LIN {X 125.150,Y 42.862,Z -41.660,A 90.000,B 90.000,C 0.000} C_DIS
LIN {X 125.083,Y 42.862,Z -40.727,A 90.000,B 90.000,C 0.000} C_DIS
LIN {X 124.959,Y 42.862,Z -39.799,A 90.000,B 90.000,C 0.000} C_DIS
LIN {X 124.777,Y 42.862,Z -38.880,A 90.000,B 90.000,C 0.000} C_DIS
LIN {X 124.742,Y 42.862,Z -38.744,A 90.000,B 90.000,C 0.000} C_DIS
LIN {X 144.015,Y 42.862,Z -38.744,A 90.000,B 90.000,C 0.000} C_DIS
LIN {X 144.015,Y 42.862,Z -31.195,A 90.000,B 90.000,C 0.000} C_DIS
LIN {X 120.047,Y 42.862,Z -31.195,A 90.000,B 90.000,C 0.000} C_DIS
LIN {X 119.392,Y 42.862,Z -30.675,A 90.000,B 90.000,C 0.000} C_DIS
LIN {X 118.703,Y 42.862,Z -30.202,A 90.000,B 90.000,C 0.000} C_DIS
LIN {X 117.982,Y 42.862,Z -29.778,A 90.000,B 90.000,C 0.000} C_DIS
LIN {X 117.233,Y 42.862,Z -29.405,A 90.000,B 90.000,C 0.000} C_DIS
LIN {X 116.461,Y 42.862,Z -29.085,A 90.000,B 90.000,C 0.000} C_DIS
LIN {X 115.668,Y 42.862,Z -28.820,A 90.000,B 90.000,C 0.000} C_DIS
LIN {X 114.858,Y 42.862,Z -28.611,A 90.000,B 90.000,C 0.000} C_DIS
LIN {X 114.036,Y 42.862,Z -28.458,A 90.000,B 90.000,C 0.000} C_DIS
LIN {X 113.205,Y 42.862,Z -28.364,A 90.000,B 90.000,C 0.000} C_DIS
LIN {X 113.054,Y 42.862,Z -28.333,A 90.000,B 90.000,C 0.000} C_DIS
LIN {X 112.017,Y 42.862,Z -28.254,A 90.000,B 90.000,C 0.000} C_DIS
LIN {X 110.978,Y 42.862,Z -28.245,A 90.000,B 90.000,C 0.000} C_DIS
LIN {X 109.940,Y 42.862,Z -28.305,A 90.000,B 90.000,C 0.000} C_DIS
LIN {X 108.908,Y 42.862,Z -28.435,A 90.000,B 90.000,C 0.000} C_DIS
LIN {X 107.888,Y 42.862,Z -28.633,A 90.000,B 90.000,C 0.000} C_DIS
LIN {X 106.883,Y 42.862,Z -28.899,A 90.000,B 90.000,C 0.000} C_DIS
LIN {X 105.898,Y 42.862,Z -29.232,A 90.000,B 90.000,C 0.000} C_DIS
LIN {X 104.937,Y 42.862,Z -29.630,A 90.000,B 90.000,C 0.000} C_DIS
LIN {X 104.006,Y 42.862,Z -30.091,A 90.000,B 90.000,C 0.000} C_DIS
LIN {X 103.107,Y 42.862,Z -30.614,A 90.000,B 90.000,C 0.000} C_DIS
LIN {X 102.245,Y 42.862,Z -31.195,A 90.000,B 90.000,C 0.000} C_DIS
LIN {X -144.015,Y 42.862,Z -31.195,A 90.000,B 90.000,C 0.000} C_DIS
LIN {X -144.015,Y 42.862,Z -38.744,A 90.000,B 90.000,C 0.000} C_DIS
LIN {X 94.730,Y 42.862,Z -38.744,A 90.000,B 90.000,C 0.000} C_DIS
LIN {X 86.696,Y 42.862,Z -46.293,A 90.000,B 90.000,C 0.000} C_DIS
LIN {X 56.285,Y 42.862,Z -46.293,A 90.000,B 90.000,C 0.000} C_DIS
LIN {X 57.224,Y 42.862,Z -46.739,A 90.000,B 90.000,C 0.000} C_DIS
LIN {X 58.135,Y 42.862,Z -47.241,A 90.000,B 90.000,C 0.000} C_DIS
LIN {X 59.013,Y 42.862,Z -47.797,A 90.000,B 90.000,C 0.000} C_DIS
LIN {X 59.857,Y 42.862,Z -48.404,A 90.000,B 90.000,C 0.000} C_DIS
LIN {X 60.662,Y 42.862,Z -49.062,A 90.000,B 90.000,C 0.000} C_DIS
LIN {X 61.427,Y 42.862,Z -49.766,A 90.000,B 90.000,C 0.000} C_DIS
LIN {X 62.148,Y 42.862,Z -50.516,A 90.000,B 90.000,C 0.000} C_DIS
LIN {X 62.822,Y 42.862,Z -51.307,A 90.000,B 90.000,C 0.000} C_DIS
LIN {X 63.559,Y 42.862,Z -52.125,A 90.000,B 90.000,C 0.000} C_DIS
LIN {X 64.266,Y 42.862,Z -52.970,A 90.000,B 90.000,C 0.000} C_DIS
LIN {X 64.941,Y 42.862,Z -53.841,A 90.000,B 90.000,C 0.000} C_DIS
LIN {X 78.905,Y 42.862,Z -53.841,A 90.000,B 90.000,C 0.000} C_DIS
LIN {X 77.974,Y 42.862,Z -55.025,A 90.000,B 90.000,C 0.000} C_DIS
LIN {X 77.084,Y 42.862,Z -56.241,A 90.000,B 90.000,C 0.000} C_DIS
LIN {X 76.237,Y 42.862,Z -57.487,A 90.000,B 90.000,C 0.000} C_DIS
LIN {X 75.433,Y 42.862,Z -58.761,A 90.000,B 90.000,C 0.000} C_DIS
LIN {X 74.674,Y 42.862,Z -60.063,A 90.000,B 90.000,C 0.000} C_DIS
LIN {X 73.961,Y 42.862,Z -61.390,A 90.000,B 90.000,C 0.000} C_DIS
LIN {X 69.034,Y 42.862,Z -61.390,A 90.000,B 90.000,C 0.000} C_DIS
LIN {X 68.549,Y 42.862,Z -60.157,A 90.000,B 90.000,C 0.000} C_DIS
LIN {X 68.010,Y 42.862,Z -58.947,A 90.000,B 90.000,C 0.000} C_DIS
LIN {X 67.418,Y 42.862,Z -57.762,A 90.000,B 90.000,C 0.000} C_DIS
LIN {X 66.774,Y 42.862,Z -56.605,A 90.000,B 90.000,C 0.000} C_DIS
LIN {X 66.080,Y 42.862,Z -55.477,A 90.000,B 90.000,C 0.000} C_DIS
LIN {X 65.335,Y 42.862,Z -54.381,A 90.000,B 90.000,C 0.000} C_DIS
LIN {X 64.543,Y 42.862,Z -53.320,A 90.000,B 90.000,C 0.000} C_DIS
LIN {X 63.705,Y 42.862,Z -52.294,A 90.000,B 90.000,C 0.000} C_DIS
LIN {X 62.822,Y 42.862,Z -51.307,A 90.000,B 90.000,C 0.000} C_DIS
LIN {X 62.102,Y 42.862,Z -50.466,A 90.000,B 90.000,C 0.000} C_DIS
LIN {X 61.330,Y 42.862,Z -49.672,A 90.000,B 90.000,C 0.000} C_DIS
LIN {X 60.509,Y 42.862,Z -48.930,A 90.000,B 90.000,C 0.000} C_DIS
LIN {X 59.641,Y 42.862,Z -48.241,A 90.000,B 90.000,C 0.000} C_DIS
LIN {X 58.732,Y 42.862,Z -47.610,A 90.000,B 90.000,C 0.000} C_DIS
LIN {X 57.783,Y 42.862,Z -47.039,A 90.000,B 90.000,C 0.000} C_DIS
LIN {X 56.800,Y 42.862,Z -46.529,A 90.000,B 90.000,C 0.000} C_DIS
LIN {X 55.787,Y 42.862,Z -46.083,A 90.000,B 90.000,C 0.000} C_DIS
LIN {X 54.746,Y 42.862,Z -45.704,A 90.000,B 90.000,C 0.000} C_DIS
LIN {X 53.684,Y 42.862,Z -45.392,A 90.000,B 90.000,C 0.000} C_DIS
LIN {X 52.797,Y 42.862,Z -45.129,A 90.000,B 90.000,C 0.000} C_DIS
LIN {X 51.895,Y 42.862,Z -44.923,A 90.000,B 90.000,C 0.000} C_DIS
LIN {X 50.982,Y 42.862,Z -44.775,A 90.000,B 90.000,C 0.000} C_DIS
LIN {X 50.062,Y 42.862,Z -44.685,A 90.000,B 90.000,C 0.000} C_DIS
LIN {X 49.137,Y 42.862,Z -44.654,A 90.000,B 90.000,C 0.000} C_DIS
LIN {X 48.213,Y 42.862,Z -44.681,A 90.000,B 90.000,C 0.000} C_DIS
LIN {X 47.292,Y 42.862,Z -44.767,A 90.000,B 90.000,C 0.000} C_DIS
LIN {X 46.319,Y 42.862,Z -44.277,A 90.000,B 90.000,C 0.000} C_DIS
LIN {X 45.314,Y 42.862,Z -43.856,A 90.000,B 90.000,C 0.000} C_DIS
LIN {X 44.282,Y 42.862,Z -43.505,A 90.000,B 90.000,C 0.000} C_DIS
LIN {X 43.229,Y 42.862,Z -43.227,A 90.000,B 90.000,C 0.000} C_DIS
LIN {X 42.159,Y 42.862,Z -43.022,A 90.000,B 90.000,C 0.000} C_DIS
LIN {X 41.077,Y 42.862,Z -42.891,A 90.000,B 90.000,C 0.000} C_DIS
LIN {X 39.989,Y 42.862,Z -42.836,A 90.000,B 90.000,C 0.000} C_DIS
LIN {X 38.899,Y 42.862,Z -42.856,A 90.000,B 90.000,C 0.000} C_DIS
LIN {X 37.814,Y 42.862,Z -42.951,A 90.000,B 90.000,C 0.000} C_DIS
LIN {X 36.738,Y 42.862,Z -43.121,A 90.000,B 90.000,C 0.000} C_DIS
LIN {X 35.676,Y 42.862,Z -43.365,A 90.000,B 90.000,C 0.000} C_DIS
LIN {X 34.633,Y 42.862,Z -43.681,A 90.000,B 90.000,C 0.000} C_DIS
LIN {X 33.615,Y 42.862,Z -44.069,A 90.000,B 90.000,C 0.000} C_DIS
LIN {X 32.626,Y 42.862,Z -44.527,A 90.000,B 90.000,C 0.000} C_DIS
LIN {X 31.671,Y 42.862,Z -45.052,A 90.000,B 90.000,C 0.000} C_DIS
LIN {X 30.755,Y 42.862,Z -45.641,A 90.000,B 90.000,C 0.000} C_DIS
LIN {X 29.882,Y 42.862,Z -46.293,A 90.000,B 90.000,C 0.000} C_DIS
LIN {X -144.015,Y 42.862,Z -46.293,A 90.000,B 90.000,C 0.000} C_DIS
LIN {X -144.015,Y 42.862,Z -53.841,A 90.000,B 90.000,C 0.000} C_DIS
LIN {X 24.711,Y 42.862,Z -53.841,A 90.000,B 90.000,C 0.000} C_DIS
LIN {X 24.711,Y 42.862,Z -53.843,A 90.000,B 90.000,C 0.000} C_DIS
LIN {X 24.175,Y 42.862,Z -54.360,A 90.000,B 90.000,C 0.000} C_DIS
LIN {X 23.668,Y 42.862,Z -54.907,A 90.000,B 90.000,C 0.000} C_DIS
LIN {X 23.192,Y 42.862,Z -55.480,A 90.000,B 90.000,C 0.000} C_DIS
LIN {X 22.748,Y 42.862,Z -56.078,A 90.000,B 90.000,C 0.000} C_DIS
LIN {X 22.337,Y 42.862,Z -56.700,A 90.000,B 90.000,C 0.000} C_DIS
LIN {X 21.899,Y 42.862,Z -57.594,A 90.000,B 90.000,C 0.000} C_DIS
LIN {X 21.518,Y 42.862,Z -58.513,A 90.000,B 90.000,C 0.000} C_DIS
LIN {X 21.196,Y 42.862,Z -59.455,A 90.000,B 90.000,C 0.000} C_DIS
LIN {X 20.934,Y 42.862,Z -60.415,A 90.000,B 90.000,C 0.000} C_DIS
LIN {X 20.734,Y 42.862,Z -61.390,A 90.000,B 90.000,C 0.000} C_DIS
LIN {X -144.015,Y 42.862,Z -61.390,A 90.000,B 90.000,C 0.000} C_DIS
LIN {X -144.015,Y 42.862,Z -68.939,A 90.000,B 90.000,C 0.000} C_DIS
LIN {X -16.258,Y 42.862,Z -68.939,A 90.000,B 90.000,C 0.000} C_DIS
LIN {X -17.508,Y 42.862,Z -69.258,A 90.000,B 90.000,C 0.000} C_DIS
LIN {X -18.739,Y 42.862,Z -69.643,A 90.000,B 90.000,C 0.000} C_DIS
LIN {X -19.948,Y 42.862,Z -70.093,A 90.000,B 90.000,C 0.000} C_DIS
LIN {X -21.131,Y 42.862,Z -70.607,A 90.000,B 90.000,C 0.000} C_DIS
LIN {X -22.284,Y 42.862,Z -71.183,A 90.000,B 90.000,C 0.000} C_DIS
LIN {X -23.406,Y 42.862,Z -71.821,A 90.000,B 90.000,C 0.000} C_DIS
LIN {X -24.492,Y 42.862,Z -72.517,A 90.000,B 90.000,C 0.000} C_DIS
LIN {X -25.539,Y 42.862,Z -73.271,A 90.000,B 90.000,C 0.000} C_DIS
LIN {X -26.544,Y 42.862,Z -74.079,A 90.000,B 90.000,C 0.000} C_DIS
LIN {X -27.504,Y 42.862,Z -74.940,A 90.000,B 90.000,C 0.000} C_DIS
LIN {X -28.266,Y 42.862,Z -75.705,A 90.000,B 90.000,C 0.000} C_DIS
LIN {X -29.009,Y 42.862,Z -76.488,A 90.000,B 90.000,C 0.000} C_DIS
LIN {X -144.015,Y 42.862,Z -76.488,A 90.000,B 90.000,C 0.000} C_DIS
LIN {X -144.015,Y 42.862,Z -84.037,A 90.000,B 90.000,C 0.000} C_DIS
LIN {X -34.671,Y 42.862,Z -84.037,A 90.000,B 90.000,C 0.000} C_DIS
LIN {X -35.506,Y 42.862,Z -85.491,A 90.000,B 90.000,C 0.000} C_DIS
LIN {X -36.286,Y 42.862,Z -86.975,A 90.000,B 90.000,C 0.000} C_DIS
LIN {X -37.012,Y 42.862,Z -88.487,A 90.000,B 90.000,C 0.000} C_DIS
LIN {X -37.681,Y 42.862,Z -90.025,A 90.000,B 90.000,C 0.000} C_DIS
LIN {X -38.293,Y 42.862,Z -91.586,A 90.000,B 90.000,C 0.000} C_DIS
LIN {X -144.015,Y 42.862,Z -91.586,A 90.000,B 90.000,C 0.000} C_DIS
LIN {X -144.015,Y 42.862,Z -99.134,A 90.000,B 90.000,C 0.000} C_DIS
LIN {X -40.372,Y 42.862,Z -99.134,A 90.000,B 90.000,C 0.000} C_DIS
LIN {X -40.520,Y 42.862,Z -99.983,A 90.000,B 90.000,C 0.000} C_DIS
LIN {X -40.653,Y 42.862,Z -100.835,A 90.000,B 90.000,C 0.000} C_DIS
LIN {X -40.931,Y 42.862,Z -101.987,A 90.000,B 90.000,C 0.000} C_DIS
LIN {X -41.159,Y 42.862,Z -103.150,A 90.000,B 90.000,C 0.000} C_DIS
LIN {X -41.337,Y 42.862,Z -104.322,A 90.000,B 90.000,C 0.000} C_DIS
LIN {X -41.464,Y 42.862,Z -105.500,A 90.000,B 90.000,C 0.000} C_DIS
LIN {X -41.540,Y 42.862,Z -106.683,A 90.000,B 90.000,C 0.000} C_DIS
LIN {X -144.015,Y 42.862,Z -106.683,A 90.000,B 90.000,C 0.000} C_DIS
LIN {X -144.015,Y 42.862,Z -114.232,A 90.000,B 90.000,C 0.000} C_DIS
LIN {X -41.253,Y 42.862,Z -114.232,A 90.000,B 90.000,C 0.000} C_DIS
LIN {X -41.121,Y 42.862,Z -114.920,A 90.000,B 90.000,C 0.000} C_DIS
LIN {X -40.964,Y 42.862,Z -115.603,A 90.000,B 90.000,C 0.000} C_DIS
LIN {X -40.701,Y 42.862,Z -116.533,A 90.000,B 90.000,C 0.000} C_DIS
LIN {X -40.478,Y 42.862,Z -117.474,A 90.000,B 90.000,C 0.000} C_DIS
LIN {X -40.295,Y 42.862,Z -118.423,A 90.000,B 90.000,C 0.000} C_DIS
LIN {X -40.153,Y 42.862,Z -119.379,A 90.000,B 90.000,C 0.000} C_DIS
LIN {X -40.093,Y 42.862,Z -119.584,A 90.000,B 90.000,C 0.000} C_DIS
LIN {X -40.057,Y 42.862,Z -119.773,A 90.000,B 90.000,C 0.000} C_DIS
LIN {X -39.705,Y 42.862,Z -120.775,A 90.000,B 90.000,C 0.000} C_DIS
LIN {X -39.361,Y 42.862,Z -121.781,A 90.000,B 90.000,C 0.000} C_DIS
LIN {X -144.015,Y 42.862,Z -121.781,A 90.000,B 90.000,C 0.000} C_DIS
LIN {X -144.015,Y 42.862,Z -129.329,A 90.000,B 90.000,C 0.000} C_DIS
LIN {X -36.708,Y 42.862,Z -129.329,A 90.000,B 90.000,C 0.000} C_DIS
LIN {X -36.411,Y 42.862,Z -129.970,A 90.000,B 90.000,C 0.000} C_DIS
LIN {X -36.089,Y 42.862,Z -130.598,A 90.000,B 90.000,C 0.000} C_DIS
LIN {X -35.628,Y 42.862,Z -131.888,A 90.000,B 90.000,C 0.000} C_DIS
LIN {X -35.126,Y 42.862,Z -133.162,A 90.000,B 90.000,C 0.000} C_DIS
LIN {X -34.584,Y 42.862,Z -134.419,A 90.000,B 90.000,C 0.000} C_DIS
LIN {X -34.001,Y 42.862,Z -135.658,A 90.000,B 90.000,C 0.000} C_DIS
LIN {X -33.379,Y 42.862,Z -136.878,A 90.000,B 90.000,C 0.000} C_DIS
LIN {X -144.015,Y 42.862,Z -136.878,A 90.000,B 90.000,C 0.000} C_DIS
LIN {X -144.015,Y 42.862,Z -144.427,A 90.000,B 90.000,C 0.000} C_DIS
LIN {X -28.091,Y 42.862,Z -144.427,A 90.000,B 90.000,C 0.000} C_DIS
LIN {X -26.928,Y 42.862,Z -145.648,A 90.000,B 90.000,C 0.000} C_DIS
LIN {X -25.719,Y 42.862,Z -146.824,A 90.000,B 90.000,C 0.000} C_DIS
LIN {X -24.467,Y 42.862,Z -147.953,A 90.000,B 90.000,C 0.000} C_DIS
LIN {X -23.173,Y 42.862,Z -149.035,A 90.000,B 90.000,C 0.000} C_DIS
LIN {X -21.839,Y 42.862,Z -150.066,A 90.000,B 90.000,C 0.000} C_DIS
LIN {X -20.468,Y 42.862,Z -151.047,A 90.000,B 90.000,C 0.000} C_DIS
LIN {X -19.060,Y 42.862,Z -151.976,A 90.000,B 90.000,C 0.000} C_DIS
LIN {X -144.015,Y 42.862,Z -151.976,A 90.000,B 90.000,C 0.000} C_DIS
LIN {X -144.015,Y 42.862,Z -159.525,A 90.000,B 90.000,C 0.000} C_DIS
LIN {X 24.265,Y 42.862,Z -159.525,A 90.000,B 90.000,C 0.000} C_DIS
LIN {X 23.466,Y 42.862,Z -160.862,A 90.000,B 90.000,C 0.000} C_DIS
LIN {X 22.621,Y 42.862,Z -162.169,A 90.000,B 90.000,C 0.000} C_DIS
LIN {X 21.729,Y 42.862,Z -163.445,A 90.000,B 90.000,C 0.000} C_DIS
LIN {X 20.793,Y 42.862,Z -164.689,A 90.000,B 90.000,C 0.000} C_DIS
LIN {X 19.813,Y 42.862,Z -165.899,A 90.000,B 90.000,C 0.000} C_DIS
LIN {X 18.790,Y 42.862,Z -167.073,A 90.000,B 90.000,C 0.000} C_DIS
LIN {X -144.015,Y 42.862,Z -167.073,A 90.000,B 90.000,C 0.000} C_DIS
LIN {X -144.015,Y 42.862,Z -174.622,A 90.000,B 90.000,C 0.000} C_DIS
LIN {X 10.993,Y 42.862,Z -174.622,A 90.000,B 90.000,C 0.000} C_DIS
LIN {X 9.938,Y 42.862,Z -175.710,A 90.000,B 90.000,C 0.000} C_DIS
LIN {X 8.046,Y 42.862,Z -177.766,A 90.000,B 90.000,C 0.000} C_DIS
LIN {X 6.126,Y 42.862,Z -179.795,A 90.000,B 90.000,C 0.000} C_DIS
LIN {X 5.088,Y 42.862,Z -180.989,A 90.000,B 90.000,C 0.000} C_DIS
LIN {X 4.035,Y 42.862,Z -182.171,A 90.000,B 90.000,C 0.000} C_DIS
LIN {X -144.015,Y 42.862,Z -182.171,A 90.000,B 90.000,C 0.000} C_DIS
LIN {X -144.015,Y 42.862,Z -189.720,A 90.000,B 90.000,C 0.000} C_DIS
LIN {X -3.333,Y 42.862,Z -189.720,A 90.000,B 90.000,C 0.000} C_DIS
LIN {X -4.736,Y 42.862,Z -191.028,A 90.000,B 90.000,C 0.000} C_DIS
LIN {X -6.158,Y 42.862,Z -192.316,A 90.000,B 90.000,C 0.000} C_DIS
LIN {X -8.323,Y 42.862,Z -194.009,A 90.000,B 90.000,C 0.000} C_DIS
LIN {X -10.520,Y 42.862,Z -195.660,A 90.000,B 90.000,C 0.000} C_DIS
LIN {X -12.749,Y 42.862,Z -197.269,A 90.000,B 90.000,C 0.000} C_DIS
LIN {X -144.015,Y 42.862,Z -197.269,A 90.000,B 90.000,C 0.000} C_DIS
LIN {X -144.015,Y 42.862,Z -204.817,A 90.000,B 90.000,C 0.000} C_DIS
LIN {X -24.715,Y 42.862,Z -204.817,A 90.000,B 90.000,C 0.000} C_DIS
LIN {X -28.376,Y 42.862,Z -206.710,A 90.000,B 90.000,C 0.000} C_DIS
LIN {X -32.061,Y 42.862,Z -208.555,A 90.000,B 90.000,C 0.000} C_DIS
LIN {X -35.770,Y 42.862,Z -210.351,A 90.000,B 90.000,C 0.000} C_DIS
LIN {X -39.503,Y 42.862,Z -212.098,A 90.000,B 90.000,C 0.000} C_DIS
LIN {X -40.093,Y 42.862,Z -212.366,A 90.000,B 90.000,C 0.000} C_DIS
LIN {X -144.015,Y 42.862,Z -212.366,A 90.000,B 90.000,C 0.000} C_DIS
LIN {X -144.015,Y 42.862,Z -219.915,A 90.000,B 90.000,C 0.000} C_DIS
LIN {X -55.981,Y 42.862,Z -219.915,A 90.000,B 90.000,C 0.000} C_DIS
LIN {X -60.909,Y 42.862,Z -222.383,A 90.000,B 90.000,C 0.000} C_DIS
LIN {X -65.811,Y 42.862,Z -224.899,A 90.000,B 90.000,C 0.000} C_DIS
LIN {X -70.689,Y 42.862,Z -227.464,A 90.000,B 90.000,C 0.000} C_DIS
LIN {X -144.015,Y 42.862,Z -227.464,A 90.000,B 90.000,C 0.000} C_DIS
LIN {X -144.015,Y 42.862,Z -235.012,A 90.000,B 90.000,C 0.000} C_DIS
LIN {X -84.330,Y 42.862,Z -235.012,A 90.000,B 90.000,C 0.000} C_DIS
LIN {X -86.708,Y 42.862,Z -236.453,A 90.000,B 90.000,C 0.000} C_DIS
LIN {X -89.064,Y 42.862,Z -237.928,A 90.000,B 90.000,C 0.000} C_DIS
LIN {X -91.399,Y 42.862,Z -239.438,A 90.000,B 90.000,C 0.000} C_DIS
LIN {X -93.711,Y 42.862,Z -240.983,A 90.000,B 90.000,C 0.000} C_DIS
LIN {X -96.000,Y 42.862,Z -242.561,A 90.000,B 90.000,C 0.000} C_DIS
LIN {X -144.015,Y 42.862,Z -242.561,A 90.000,B 90.000,C 0.000} C_DIS
LIN {X -144.015,Y 42.862,Z -23.646,A 90.000,B 90.000,C 0.000} C_DIS
LIN {X 144.015,Y 42.862,Z -23.646,A 90.000,B 90.000,C 0.000} C_DIS
LIN {X 144.015,Y 42.862,Z -16.098,A 90.000,B 90.000,C 0.000} C_DIS
LIN {X -144.015,Y 42.862,Z -16.098,A 90.000,B 90.000,C 0.000} C_DIS
LIN {X -144.015,Y 42.862,Z -8.549,A 90.000,B 90.000,C 0.000} C_DIS
LIN {X 144.015,Y 42.862,Z -8.549,A 90.000,B 90.000,C 0.000} C_DIS
LIN {X 144.015,Y 42.862,Z -1.000,A 90.000,B 90.000,C 0.000} C_DIS
LIN {X -144.015,Y 42.862,Z -1.000,A 90.000,B 90.000,C 0.000} C_DIS
LIN {X -3.685,Y 42.862,Z -68.939,A 90.000,B 90.000,C 0.000} C_DIS
LIN {X 10.592,Y 42.862,Z -68.939,A 90.000,B 90.000,C 0.000} C_DIS
LIN {X 10.606,Y 42.862,Z -73.107,A 90.000,B 90.000,C 0.000} C_DIS
LIN {X 7.736,Y 42.862,Z -72.365,A 90.000,B 90.000,C 0.000} C_DIS
LIN {X 4.853,Y 42.862,Z -71.676,A 90.000,B 90.000,C 0.000} C_DIS
LIN {X 1.958,Y 42.862,Z -71.039,A 90.000,B 90.000,C 0.000} C_DIS
LIN {X -0.948,Y 42.862,Z -70.455,A 90.000,B 90.000,C 0.000} C_DIS
LIN {X -3.864,Y 42.862,Z -69.924,A 90.000,B 90.000,C 0.000} C_DIS
LIN {X -4.992,Y 42.862,Z -69.694,A 90.000,B 90.000,C 0.000} C_DIS
LIN {X -6.128,Y 42.862,Z -69.514,A 90.000,B 90.000,C 0.000} C_DIS
LIN {X -7.272,Y 42.862,Z -69.383,A 90.000,B 90.000,C 0.000} C_DIS
LIN {X -8.420,Y 42.862,Z -69.302,A 90.000,B 90.000,C 0.000} C_DIS
LIN {X -9.570,Y 42.862,Z -69.272,A 90.000,B 90.000,C 0.000} C_DIS
LIN {X -10.721,Y 42.862,Z -69.292,A 90.000,B 90.000,C 0.000} C_DIS
LIN {X -11.870,Y 42.862,Z -69.361,A 90.000,B 90.000,C 0.000} C_DIS
LIN {X -13.141,Y 42.862,Z -69.448,A 90.000,B 90.000,C 0.000} C_DIS
LIN {X -14.406,Y 42.862,Z -69.605,A 90.000,B 90.000,C 0.000} C_DIS
LIN {X -15.659,Y 42.862,Z -69.832,A 90.000,B 90.000,C 0.000} C_DIS
LIN {X -16.899,Y 42.862,Z -70.127,A 90.000,B 90.000,C 0.000} C_DIS
LIN {X -18.120,Y 42.862,Z -70.490,A 90.000,B 90.000,C 0.000} C_DIS
LIN {X -19.320,Y 42.862,Z -70.919,A 90.000,B 90.000,C 0.000} C_DIS
LIN {X -20.494,Y 42.862,Z -71.414,A 90.000,B 90.000,C 0.000} C_DIS
LIN {X -21.639,Y 42.862,Z -71.973,A 90.000,B 90.000,C 0.000} C_DIS
LIN {X -22.752,Y 42.862,Z -72.594,A 90.000,B 90.000,C 0.000} C_DIS
LIN {X -23.828,Y 42.862,Z -73.276,A 90.000,B 90.000,C 0.000} C_DIS
LIN {X -24.866,Y 42.862,Z -74.015,A 90.000,B 90.000,C 0.000} C_DIS
LIN {X -25.861,Y 42.862,Z -74.811,A 90.000,B 90.000,C 0.000} C_DIS
LIN {X -26.811,Y 42.862,Z -75.660,A 90.000,B 90.000,C 0.000} C_DIS
LIN {X -28.077,Y 42.862,Z -76.954,A 90.000,B 90.000,C 0.000} C_DIS
LIN {X -29.289,Y 42.862,Z -78.298,A 90.000,B 90.000,C 0.000} C_DIS
LIN {X -30.445,Y 42.862,Z -79.690,A 90.000,B 90.000,C 0.000} C_DIS
LIN {X -31.543,Y 42.862,Z -81.128,A 90.000,B 90.000,C 0.000} C_DIS
LIN {X -32.583,Y 42.862,Z -82.610,A 90.000,B 90.000,C 0.000} C_DIS
LIN {X -33.561,Y 42.862,Z -84.132,A 90.000,B 90.000,C 0.000} C_DIS
LIN {X -34.476,Y 42.862,Z -85.694,A 90.000,B 90.000,C 0.000} C_DIS
LIN {X -35.327,Y 42.862,Z -87.291,A 90.000,B 90.000,C 0.000} C_DIS
LIN {X -36.112,Y 42.862,Z -88.922,A 90.000,B 90.000,C 0.000} C_DIS
LIN {X -36.830,Y 42.862,Z -90.583,A 90.000,B 90.000,C 0.000} C_DIS
LIN {X -37.480,Y 42.862,Z -92.272,A 90.000,B 90.000,C 0.000} C_DIS
LIN {X -38.060,Y 42.862,Z -93.986,A 90.000,B 90.000,C 0.000} C_DIS
LIN {X -38.570,Y 42.862,Z -95.723,A 90.000,B 90.000,C 0.000} C_DIS
LIN {X -39.009,Y 42.862,Z -97.478,A 90.000,B 90.000,C 0.000} C_DIS
LIN {X -39.377,Y 42.862,Z -99.250,A 90.000,B 90.000,C 0.000} C_DIS
LIN {X -39.671,Y 42.862,Z -101.036,A 90.000,B 90.000,C 0.000} C_DIS
LIN {X -39.961,Y 42.862,Z -102.237,A 90.000,B 90.000,C 0.000} C_DIS
LIN {X -40.195,Y 42.862,Z -103.450,A 90.000,B 90.000,C 0.000} C_DIS
LIN {X -40.372,Y 42.862,Z -104.673,A 90.000,B 90.000,C 0.000} C_DIS
LIN {X -40.492,Y 42.862,Z -105.902,A 90.000,B 90.000,C 0.000} C_DIS
LIN {X -40.555,Y 42.862,Z -107.136,A 90.000,B 90.000,C 0.000} C_DIS
LIN {X -40.560,Y 42.862,Z -108.372,A 90.000,B 90.000,C 0.000} C_DIS
LIN {X -40.508,Y 42.862,Z -109.606,A 90.000,B 90.000,C 0.000} C_DIS
LIN {X -40.546,Y 42.862,Z -110.568,A 90.000,B 90.000,C 0.000} C_DIS
LIN {X -40.534,Y 42.862,Z -111.530,A 90.000,B 90.000,C 0.000} C_DIS
LIN {X -40.474,Y 42.862,Z -112.491,A 90.000,B 90.000,C 0.000} C_DIS
LIN {X -40.364,Y 42.862,Z -113.447,A 90.000,B 90.000,C 0.000} C_DIS
LIN {X -40.206,Y 42.862,Z -114.397,A 90.000,B 90.000,C 0.000} C_DIS
LIN {X -40.000,Y 42.862,Z -115.337,A 90.000,B 90.000,C 0.000} C_DIS
LIN {X -39.734,Y 42.862,Z -116.283,A 90.000,B 90.000,C 0.000} C_DIS
LIN {X -39.506,Y 42.862,Z -117.238,A 90.000,B 90.000,C 0.000} C_DIS
LIN {X -39.319,Y 42.862,Z -118.203,A 90.000,B 90.000,C 0.000} C_DIS
LIN {X -39.171,Y 42.862,Z -119.174,A 90.000,B 90.000,C 0.000} C_DIS
LIN {X -39.119,Y 42.862,Z -119.351,A 90.000,B 90.000,C 0.000} C_DIS
LIN {X -39.089,Y 42.862,Z -119.511,A 90.000,B 90.000,C 0.000} C_DIS
LIN {X -38.572,Y 42.862,Z -120.993,A 90.000,B 90.000,C 0.000} C_DIS
LIN {X -38.075,Y 42.862,Z -122.483,A 90.000,B 90.000,C 0.000} C_DIS
LIN {X -37.597,Y 42.862,Z -123.978,A 90.000,B 90.000,C 0.000} C_DIS
LIN {X -37.537,Y 42.862,Z -124.124,A 90.000,B 90.000,C 0.000} C_DIS
LIN {X -37.324,Y 42.862,Z -124.797,A 90.000,B 90.000,C 0.000} C_DIS
LIN {X -37.062,Y 42.862,Z -125.453,A 90.000,B 90.000,C 0.000} C_DIS
LIN {X -36.753,Y 42.862,Z -126.088,A 90.000,B 90.000,C 0.000} C_DIS
LIN {X -36.523,Y 42.862,Z -126.941,A 90.000,B 90.000,C 0.000} C_DIS
LIN {X -36.248,Y 42.862,Z -127.780,A 90.000,B 90.000,C 0.000} C_DIS
LIN {X -35.931,Y 42.862,Z -128.604,A 90.000,B 90.000,C 0.000} C_DIS
LIN {X -35.571,Y 42.862,Z -129.411,A 90.000,B 90.000,C 0.000} C_DIS
LIN {X -35.169,Y 42.862,Z -130.197,A 90.000,B 90.000,C 0.000} C_DIS
LIN {X -34.647,Y 42.862,Z -131.656,A 90.000,B 90.000,C 0.000} C_DIS
LIN {X -34.070,Y 42.862,Z -133.095,A 90.000,B 90.000,C 0.000} C_DIS
LIN {X -33.441,Y 42.862,Z -134.511,A 90.000,B 90.000,C 0.000} C_DIS
LIN {X -32.759,Y 42.862,Z -135.903,A 90.000,B 90.000,C 0.000} C_DIS
LIN {X -32.026,Y 42.862,Z -137.269,A 90.000,B 90.000,C 0.000} C_DIS
LIN {X -31.243,Y 42.862,Z -138.606,A 90.000,B 90.000,C 0.000} C_DIS
LIN {X -30.411,Y 42.862,Z -139.914,A 90.000,B 90.000,C 0.000} C_DIS
LIN {X -29.530,Y 42.862,Z -141.189,A 90.000,B 90.000,C 0.000} C_DIS
LIN {X -28.431,Y 42.862,Z -142.533,A 90.000,B 90.000,C 0.000} C_DIS
LIN {X -27.280,Y 42.862,Z -143.832,A 90.000,B 90.000,C 0.000} C_DIS
LIN {X -26.078,Y 42.862,Z -145.084,A 90.000,B 90.000,C 0.000} C_DIS
LIN {X -24.827,Y 42.862,Z -146.287,A 90.000,B 90.000,C 0.000} C_DIS
LIN {X -23.530,Y 42.862,Z -147.440,A 90.000,B 90.000,C 0.000} C_DIS
LIN {X -22.188,Y 42.862,Z -148.541,A 90.000,B 90.000,C 0.000} C_DIS
LIN {X -20.803,Y 42.862,Z -149.587,A 90.000,B 90.000,C 0.000} C_DIS
LIN {X -19.378,Y 42.862,Z -150.577,A 90.000,B 90.000,C 0.000} C_DIS
LIN {X -17.914,Y 42.862,Z -151.511,A 90.000,B 90.000,C 0.000} C_DIS
LIN {X -16.415,Y 42.862,Z -152.385,A 90.000,B 90.000,C 0.000} C_DIS
LIN {X -14.882,Y 42.862,Z -153.199,A 90.000,B 90.000,C 0.000} C_DIS
LIN {X -13.318,Y 42.862,Z -153.952,A 90.000,B 90.000,C 0.000} C_DIS
LIN {X -11.725,Y 42.862,Z -154.641,A 90.000,B 90.000,C 0.000} C_DIS
LIN {X -10.106,Y 42.862,Z -155.267,A 90.000,B 90.000,C 0.000} C_DIS
LIN {X -8.722,Y 42.862,Z -155.765,A 90.000,B 90.000,C 0.000} C_DIS
LIN {X -7.318,Y 42.862,Z -156.206,A 90.000,B 90.000,C 0.000} C_DIS
LIN {X -5.896,Y 42.862,Z -156.587,A 90.000,B 90.000,C 0.000} C_DIS
LIN {X -4.461,Y 42.862,Z -156.910,A 90.000,B 90.000,C 0.000} C_DIS
LIN {X -3.013,Y 42.862,Z -157.172,A 90.000,B 90.000,C 0.000} C_DIS
LIN {X -1.555,Y 42.862,Z -157.374,A 90.000,B 90.000,C 0.000} C_DIS
LIN {X -0.091,Y 42.862,Z -157.515,A 90.000,B 90.000,C 0.000} C_DIS
LIN {X 1.379,Y 42.862,Z -157.595,A 90.000,B 90.000,C 0.000} C_DIS
LIN {X 2.850,Y 42.862,Z -157.615,A 90.000,B 90.000,C 0.000} C_DIS
LIN {X 4.795,Y 42.862,Z -157.543,A 90.000,B 90.000,C 0.000} C_DIS
LIN {X 6.736,Y 42.862,Z -157.405,A 90.000,B 90.000,C 0.000} C_DIS
LIN {X 8.671,Y 42.862,Z -157.201,A 90.000,B 90.000,C 0.000} C_DIS
LIN {X 10.598,Y 42.862,Z -156.933,A 90.000,B 90.000,C 0.000} C_DIS
LIN {X 12.516,Y 42.862,Z -156.600,A 90.000,B 90.000,C 0.000} C_DIS
LIN {X 14.420,Y 42.862,Z -156.202,A 90.000,B 90.000,C 0.000} C_DIS
LIN {X 16.311,Y 42.862,Z -155.740,A 90.000,B 90.000,C 0.000} C_DIS
LIN {X 18.184,Y 42.862,Z -155.214,A 90.000,B 90.000,C 0.000} C_DIS
LIN {X 20.039,Y 42.862,Z -154.626,A 90.000,B 90.000,C 0.000} C_DIS
LIN {X 21.873,Y 42.862,Z -153.975,A 90.000,B 90.000,C 0.000} C_DIS
LIN {X 23.684,Y 42.862,Z -153.263,A 90.000,B 90.000,C 0.000} C_DIS
LIN {X 25.470,Y 42.862,Z -152.490,A 90.000,B 90.000,C 0.000} C_DIS
LIN {X 29.996,Y 42.862,Z -150.077,A 90.000,B 90.000,C 0.000} C_DIS
LIN {X 29.921,Y 42.862,Z -150.256,A 90.000,B 90.000,C 0.000} C_DIS
LIN {X 29.378,Y 42.862,Z -151.711,A 90.000,B 90.000,C 0.000} C_DIS
LIN {X 28.788,Y 42.862,Z -153.147,A 90.000,B 90.000,C 0.000} C_DIS
LIN {X 28.151,Y 42.862,Z -154.564,A 90.000,B 90.000,C 0.000} C_DIS
LIN {X 27.468,Y 42.862,Z -155.958,A 90.000,B 90.000,C 0.000} C_DIS
LIN {X 26.739,Y 42.862,Z -157.329,A 90.000,B 90.000,C 0.000} C_DIS
LIN {X 25.965,Y 42.862,Z -158.676,A 90.000,B 90.000,C 0.000} C_DIS
LIN {X 25.148,Y 42.862,Z -159.996,A 90.000,B 90.000,C 0.000} C_DIS
LIN {X 24.272,Y 42.862,Z -161.460,A 90.000,B 90.000,C 0.000} C_DIS
LIN {X 23.341,Y 42.862,Z -162.889,A 90.000,B 90.000,C 0.000} C_DIS
LIN {X 22.357,Y 42.862,Z -164.282,A 90.000,B 90.000,C 0.000} C_DIS
LIN {X 21.320,Y 42.862,Z -165.636,A 90.000,B 90.000,C 0.000} C_DIS
LIN {X 20.232,Y 42.862,Z -166.950,A 90.000,B 90.000,C 0.000} C_DIS
LIN {X 19.095,Y 42.862,Z -168.221,A 90.000,B 90.000,C 0.000} C_DIS
LIN {X 16.935,Y 42.862,Z -170.208,A 90.000,B 90.000,C 0.000} C_DIS
LIN {X 14.810,Y 42.862,Z -172.233,A 90.000,B 90.000,C 0.000} C_DIS
LIN {X 12.722,Y 42.862,Z -174.295,A 90.000,B 90.000,C 0.000} C_DIS
LIN {X 10.669,Y 42.862,Z -176.393,A 90.000,B 90.000,C 0.000} C_DIS
LIN {X 8.782,Y 42.862,Z -178.443,A 90.000,B 90.000,C 0.000} C_DIS
LIN {X 6.866,Y 42.862,Z -180.467,A 90.000,B 90.000,C 0.000} C_DIS
LIN {X 4.920,Y 42.862,Z -182.681,A 90.000,B 90.000,C 0.000} C_DIS
LIN {X 2.926,Y 42.862,Z -184.852,A 90.000,B 90.000,C 0.000} C_DIS
LIN {X 0.885,Y 42.862,Z -186.979,A 90.000,B 90.000,C 0.000} C_DIS
LIN {X -1.203,Y 42.862,Z -189.059,A 90.000,B 90.000,C 0.000} C_DIS
LIN {X -3.336,Y 42.862,Z -191.094,A 90.000,B 90.000,C 0.000} C_DIS
LIN {X -5.513,Y 42.862,Z -193.081,A 90.000,B 90.000,C 0.000} C_DIS
LIN {X -7.936,Y 42.862,Z -194.972,A 90.000,B 90.000,C 0.000} C_DIS
LIN {X -10.398,Y 42.862,Z -196.811,A 90.000,B 90.000,C 0.000} C_DIS
LIN {X -12.900,Y 42.862,Z -198.597,A 90.000,B 90.000,C 0.000} C_DIS
LIN {X -15.440,Y 42.862,Z -200.328,A 90.000,B 90.000,C 0.000} C_DIS
LIN {X -18.016,Y 42.862,Z -202.004,A 90.000,B 90.000,C 0.000} C_DIS
LIN {X -20.628,Y 42.862,Z -203.624,A 90.000,B 90.000,C 0.000} C_DIS
LIN {X -23.274,Y 42.862,Z -205.188,A 90.000,B 90.000,C 0.000} C_DIS
LIN {X -26.401,Y 42.862,Z -206.823,A 90.000,B 90.000,C 0.000} C_DIS
LIN {X -29.546,Y 42.862,Z -208.423,A 90.000,B 90.000,C 0.000} C_DIS
LIN {X -32.709,Y 42.862,Z -209.987,A 90.000,B 90.000,C 0.000} C_DIS
LIN {X -35.890,Y 42.862,Z -211.515,A 90.000,B 90.000,C 0.000} C_DIS
LIN {X -39.088,Y 42.862,Z -213.007,A 90.000,B 90.000,C 0.000} C_DIS
LIN {X -44.405,Y 42.862,Z -215.458,A 90.000,B 90.000,C 0.000} C_DIS
LIN {X -49.697,Y 42.862,Z -217.964,A 90.000,B 90.000,C 0.000} C_DIS
LIN {X -54.961,Y 42.862,Z -220.526,A 90.000,B 90.000,C 0.000} C_DIS
LIN {X -60.199,Y 42.862,Z -223.144,A 90.000,B 90.000,C 0.000} C_DIS
LIN {X -65.408,Y 42.862,Z -225.816,A 90.000,B 90.000,C 0.000} C_DIS
LIN {X -70.589,Y 42.862,Z -228.543,A 90.000,B 90.000,C 0.000} C_DIS
LIN {X -75.741,Y 42.862,Z -231.325,A 90.000,B 90.000,C 0.000} C_DIS
LIN {X -78.681,Y 42.862,Z -232.919,A 90.000,B 90.000,C 0.000} C_DIS
LIN {X -81.593,Y 42.862,Z -234.566,A 90.000,B 90.000,C 0.000} C_DIS
LIN {X -84.474,Y 42.862,Z -236.264,A 90.000,B 90.000,C 0.000} C_DIS
LIN {X -87.325,Y 42.862,Z -238.013,A 90.000,B 90.000,C 0.000} C_DIS
LIN {X -90.144,Y 42.862,Z -239.813,A 90.000,B 90.000,C 0.000} C_DIS
LIN {X -92.931,Y 42.862,Z -241.663,A 90.000,B 90.000,C 0.000} C_DIS
LIN {X -95.685,Y 42.862,Z -243.561,A 90.000,B 90.000,C 0.000} C_DIS
LIN {X -145.015,Y 42.862,Z -243.561,A 90.000,B 90.000,C 0.000} C_DIS
LIN {X -145.015,Y 42.862,Z 0.000,A 90.000,B 90.000,C 0.000} C_DIS
LIN {X 145.015,Y 42.862,Z 0.000,A 90.000,B 90.000,C 0.000} C_DIS
LIN {X 145.015,Y 42.862,Z -243.561,A 90.000,B 90.000,C 0.000} C_DIS
LIN {X 60.176,Y 42.862,Z -243.561,A 90.000,B 90.000,C 0.000} C_DIS
LIN {X 62.086,Y 42.862,Z -240.150,A 90.000,B 90.000,C 0.000} C_DIS
LIN {X 63.942,Y 42.862,Z -236.710,A 90.000,B 90.000,C 0.000} C_DIS
LIN {X 65.745,Y 42.862,Z -233.242,A 90.000,B 90.000,C 0.000} C_DIS
LIN {X 67.493,Y 42.862,Z -229.745,A 90.000,B 90.000,C 0.000} C_DIS
LIN {X 69.187,Y 42.862,Z -226.222,A 90.000,B 90.000,C 0.000} C_DIS
LIN {X 70.825,Y 42.862,Z -222.673,A 90.000,B 90.000,C 0.000} C_DIS
LIN {X 72.408,Y 42.862,Z -219.099,A 90.000,B 90.000,C 0.000} C_DIS
LIN {X 73.934,Y 42.862,Z -215.500,A 90.000,B 90.000,C 0.000} C_DIS
LIN {X 75.405,Y 42.862,Z -211.878,A 90.000,B 90.000,C 0.000} C_DIS
LIN {X 76.818,Y 42.862,Z -208.234,A 90.000,B 90.000,C 0.000} C_DIS
LIN {X 78.175,Y 42.862,Z -204.568,A 90.000,B 90.000,C 0.000} C_DIS
LIN {X 79.069,Y 42.862,Z -202.298,A 90.000,B 90.000,C 0.000} C_DIS
LIN {X 79.903,Y 42.862,Z -200.006,A 90.000,B 90.000,C 0.000} C_DIS
LIN {X 80.677,Y 42.862,Z -197.693,A 90.000,B 90.000,C 0.000} C_DIS
LIN {X 81.390,Y 42.862,Z -195.361,A 90.000,B 90.000,C 0.000} C_DIS
LIN {X 82.042,Y 42.862,Z -193.010,A 90.000,B 90.000,C 0.000} C_DIS
LIN {X 82.633,Y 42.862,Z -190.644,A 90.000,B 90.000,C 0.000} C_DIS
LIN {X 83.174,Y 42.862,Z -188.150,A 90.000,B 90.000,C 0.000} C_DIS
LIN {X 83.760,Y 42.862,Z -185.666,A 90.000,B 90.000,C 0.000} C_DIS
LIN {X 84.390,Y 42.862,Z -183.192,A 90.000,B 90.000,C 0.000} C_DIS
LIN {X 85.065,Y 42.862,Z -180.731,A 90.000,B 90.000,C 0.000} C_DIS
LIN {X 85.784,Y 42.862,Z -178.282,A 90.000,B 90.000,C 0.000} C_DIS
LIN {X 86.548,Y 42.862,Z -175.847,A 90.000,B 90.000,C 0.000} C_DIS
LIN {X 87.410,Y 42.862,Z -173.328,A 90.000,B 90.000,C 0.000} C_DIS
LIN {X 88.211,Y 42.862,Z -170.790,A 90.000,B 90.000,C 0.000} C_DIS
LIN {X 88.950,Y 42.862,Z -168.232,A 90.000,B 90.000,C 0.000} C_DIS
LIN {X 89.626,Y 42.862,Z -165.658,A 90.000,B 90.000,C 0.000} C_DIS
LIN {X 90.241,Y 42.862,Z -163.068,A 90.000,B 90.000,C 0.000} C_DIS
LIN {X 90.792,Y 42.862,Z -160.464,A 90.000,B 90.000,C 0.000} C_DIS
LIN {X 91.280,Y 42.862,Z -157.847,A 90.000,B 90.000,C 0.000} C_DIS
LIN {X 91.705,Y 42.862,Z -155.219,A 90.000,B 90.000,C 0.000} C_DIS
LIN {X 92.066,Y 42.862,Z -152.582,A 90.000,B 90.000,C 0.000} C_DIS
LIN {X 92.363,Y 42.862,Z -149.936,A 90.000,B 90.000,C 0.000} C_DIS
LIN {X 92.595,Y 42.862,Z -147.285,A 90.000,B 90.000,C 0.000} C_DIS
LIN {X 92.764,Y 42.862,Z -144.628,A 90.000,B 90.000,C 0.000} C_DIS
LIN {X 92.874,Y 42.862,Z -141.092,A 90.000,B 90.000,C 0.000} C_DIS
LIN {X 93.030,Y 42.862,Z -137.558,A 90.000,B 90.000,C 0.000} C_DIS
LIN {X 93.230,Y 42.862,Z -134.026,A 90.000,B 90.000,C 0.000} C_DIS
LIN {X 93.474,Y 42.862,Z -130.497,A 90.000,B 90.000,C 0.000} C_DIS
LIN {X 93.578,Y 42.862,Z -129.332,A 90.000,B 90.000,C 0.000} C_DIS
LIN {X 93.630,Y 42.862,Z -128.163,A 90.000,B 90.000,C 0.000} C_DIS
LIN {X 93.632,Y 42.862,Z -126.994,A 90.000,B 90.000,C 0.000} C_DIS
LIN {X 93.582,Y 42.862,Z -125.825,A 90.000,B 90.000,C 0.000} C_DIS
LIN {X 93.481,Y 42.862,Z -124.660,A 90.000,B 90.000,C 0.000} C_DIS
LIN {X 93.329,Y 42.862,Z -123.500,A 90.000,B 90.000,C 0.000} C_DIS
LIN {X 93.178,Y 42.862,Z -122.870,A 90.000,B 90.000,C 0.000} C_DIS
LIN {X 93.072,Y 42.862,Z -122.231,A 90.000,B 90.000,C 0.000} C_DIS
LIN {X 93.013,Y 42.862,Z -121.586,A 90.000,B 90.000,C 0.000} C_DIS
LIN {X 92.797,Y 42.862,Z -120.745,A 90.000,B 90.000,C 0.000} C_DIS
LIN {X 92.636,Y 42.862,Z -119.891,A 90.000,B 90.000,C 0.000} C_DIS
LIN {X 92.529,Y 42.862,Z -119.029,A 90.000,B 90.000,C 0.000} C_DIS
LIN {X 92.537,Y 42.862,Z -118.894,A 90.000,B 90.000,C 0.000} C_DIS
LIN {X 92.905,Y 42.862,Z -117.894,A 90.000,B 90.000,C 0.000} C_DIS
LIN {X 93.237,Y 42.862,Z -116.882,A 90.000,B 90.000,C 0.000} C_DIS
LIN {X 93.535,Y 42.862,Z -115.859,A 90.000,B 90.000,C 0.000} C_DIS
LIN {X 93.797,Y 42.862,Z -114.827,A 90.000,B 90.000,C 0.000} C_DIS
LIN {X 93.815,Y 42.862,Z -114.731,A 90.000,B 90.000,C 0.000} C_DIS
LIN {X 94.155,Y 42.862,Z -113.391,A 90.000,B 90.000,C 0.000} C_DIS
LIN {X 94.443,Y 42.862,Z -112.365,A 90.000,B 90.000,C 0.000} C_DIS
LIN {X 94.672,Y 42.862,Z -111.324,A 90.000,B 90.000,C 0.000} C_DIS
LIN {X 94.843,Y 42.862,Z -110.272,A 90.000,B 90.000,C 0.000} C_DIS
LIN {X 94.954,Y 42.862,Z -109.212,A 90.000,B 90.000,C 0.000} C_DIS
LIN {X 95.005,Y 42.862,Z -108.147,A 90.000,B 90.000,C 0.000} C_DIS
LIN {X 94.996,Y 42.862,Z -107.082,A 90.000,B 90.000,C 0.000} C_DIS
LIN {X 94.927,Y 42.862,Z -106.018,A 90.000,B 90.000,C 0.000} C_DIS
LIN {X 94.798,Y 42.862,Z -104.960,A 90.000,B 90.000,C 0.000} C_DIS
LIN {X 95.394,Y 42.862,Z -104.269,A 90.000,B 90.000,C 0.000} C_DIS
LIN {X 95.944,Y 42.862,Z -103.542,A 90.000,B 90.000,C 0.000} C_DIS
LIN {X 96.447,Y 42.862,Z -102.781,A 90.000,B 90.000,C 0.000} C_DIS
LIN {X 96.900,Y 42.862,Z -101.989,A 90.000,B 90.000,C 0.000} C_DIS
LIN {X 97.302,Y 42.862,Z -101.170,A 90.000,B 90.000,C 0.000} C_DIS
LIN {X 97.651,Y 42.862,Z -100.327,A 90.000,B 90.000,C 0.000} C_DIS
LIN {X 97.944,Y 42.862,Z -99.463,A 90.000,B 90.000,C 0.000} C_DIS
LIN {X 98.274,Y 42.862,Z -98.143,A 90.000,B 90.000,C 0.000} C_DIS
LIN {X 98.555,Y 42.862,Z -96.811,A 90.000,B 90.000,C 0.000} C_DIS
LIN {X 98.787,Y 42.862,Z -95.470,A 90.000,B 90.000,C 0.000} C_DIS
LIN {X 98.968,Y 42.862,Z -94.122,A 90.000,B 90.000,C 0.000} C_DIS
LIN {X 99.100,Y 42.862,Z -92.767,A 90.000,B 90.000,C 0.000} C_DIS
LIN {X 100.291,Y 42.862,Z -91.854,A 90.000,B 90.000,C 0.000} C_DIS
LIN {X 101.516,Y 42.862,Z -90.705,A 90.000,B 90.000,C 0.000} C_DIS
LIN {X 102.699,Y 42.862,Z -89.513,A 90.000,B 90.000,C 0.000} C_DIS
LIN {X 103.837,Y 42.862,Z -88.279,A 90.000,B 90.000,C 0.000} C_DIS
LIN {X 104.930,Y 42.862,Z -87.004,A 90.000,B 90.000,C 0.000} C_DIS
LIN {X 105.976,Y 42.862,Z -85.690,A 90.000,B 90.000,C 0.000} C_DIS
LIN {X 106.974,Y 42.862,Z -84.340,A 90.000,B 90.000,C 0.000} C_DIS
LIN {X 107.922,Y 42.862,Z -82.954,A 90.000,B 90.000,C 0.000} C_DIS
LIN {X 108.819,Y 42.862,Z -81.534,A 90.000,B 90.000,C 0.000} C_DIS
LIN {X 109.887,Y 42.862,Z -79.545,A 90.000,B 90.000,C 0.000} C_DIS
LIN {X 110.908,Y 42.862,Z -77.531,A 90.000,B 90.000,C 0.000} C_DIS
LIN {X 111.881,Y 42.862,Z -75.494,A 90.000,B 90.000,C 0.000} C_DIS
LIN {X 112.807,Y 42.862,Z -73.435,A 90.000,B 90.000,C 0.000} C_DIS
LIN {X 113.685,Y 42.862,Z -71.354,A 90.000,B 90.000,C 0.000} C_DIS
LIN {X 114.514,Y 42.862,Z -69.254,A 90.000,B 90.000,C 0.000} C_DIS
LIN {X 115.293,Y 42.862,Z -67.135,A 90.000,B 90.000,C 0.000} C_DIS
LIN {X 116.024,Y 42.862,Z -64.999,A 90.000,B 90.000,C 0.000} C_DIS
LIN {X 116.598,Y 42.862,Z -63.108,A 90.000,B 90.000,C 0.000} C_DIS
LIN {X 117.233,Y 42.862,Z -61.236,A 90.000,B 90.000,C 0.000} C_DIS
LIN {X 117.926,Y 42.862,Z -59.386,A 90.000,B 90.000,C 0.000} C_DIS
LIN {X 118.677,Y 42.862,Z -57.558,A 90.000,B 90.000,C 0.000} C_DIS
LIN {X 119.486,Y 42.862,Z -55.755,A 90.000,B 90.000,C 0.000} C_DIS
LIN {X 120.186,Y 42.862,Z -54.498,A 90.000,B 90.000,C 0.000} C_DIS
LIN {X 120.840,Y 42.862,Z -53.216,A 90.000,B 90.000,C 0.000} C_DIS
LIN {X 121.448,Y 42.862,Z -51.912,A 90.000,B 90.000,C 0.000} C_DIS
LIN {X 122.010,Y 42.862,Z -50.587,A 90.000,B 90.000,C 0.000} C_DIS
LIN {X 122.525,Y 42.862,Z -49.243,A 90.000,B 90.000,C 0.000} C_DIS
LIN {X 122.991,Y 42.862,Z -47.882,A 90.000,B 90.000,C 0.000} C_DIS
LIN {X 123.356,Y 42.862,Z -46.957,A 90.000,B 90.000,C 0.000} C_DIS
LIN {X 123.655,Y 42.862,Z -46.008,A 90.000,B 90.000,C 0.000} C_DIS
LIN {X 123.886,Y 42.862,Z -45.040,A 90.000,B 90.000,C 0.000} C_DIS
LIN {X 124.047,Y 42.862,Z -44.059,A 90.000,B 90.000,C 0.000} C_DIS
LIN {X 124.139,Y 42.862,Z -43.068,A 90.000,B 90.000,C 0.000} C_DIS
LIN {X 124.161,Y 42.862,Z -42.074,A 90.000,B 90.000,C 0.000} C_DIS
LIN {X 124.112,Y 42.862,Z -41.080,A 90.000,B 90.000,C 0.000} C_DIS
LIN {X 123.994,Y 42.862,Z -40.093,A 90.000,B 90.000,C 0.000} C_DIS
LIN {X 123.805,Y 42.862,Z -39.116,A 90.000,B 90.000,C 0.000} C_DIS
LIN {X 123.760,Y 42.862,Z -38.939,A 90.000,B 90.000,C 0.000} C_DIS
LIN {X 123.521,Y 42.862,Z -38.048,A 90.000,B 90.000,C 0.000} C_DIS
LIN {X 123.218,Y 42.862,Z -37.176,A 90.000,B 90.000,C 0.000} C_DIS
LIN {X 122.852,Y 42.862,Z -36.329,A 90.000,B 90.000,C 0.000} C_DIS
LIN {X 122.424,Y 42.862,Z -35.512,A 90.000,B 90.000,C 0.000} C_DIS
LIN {X 121.937,Y 42.862,Z -34.727,A 90.000,B 90.000,C 0.000} C_DIS
LIN {X 121.395,Y 42.862,Z -33.981,A 90.000,B 90.000,C 0.000} C_DIS
LIN {X 120.798,Y 42.862,Z -33.277,A 90.000,B 90.000,C 0.000} C_DIS
LIN {X 120.152,Y 42.862,Z -32.618,A 90.000,B 90.000,C 0.000} C_DIS
LIN {X 119.459,Y 42.862,Z -32.009,A 90.000,B 90.000,C 0.000} C_DIS
LIN {X 118.850,Y 42.862,Z -31.518,A 90.000,B 90.000,C 0.000} C_DIS
LIN {X 118.207,Y 42.862,Z -31.072,A 90.000,B 90.000,C 0.000} C_DIS
LIN {X 117.534,Y 42.862,Z -30.673,A 90.000,B 90.000,C 0.000} C_DIS
LIN {X 116.834,Y 42.862,Z -30.323,A 90.000,B 90.000,C 0.000} C_DIS
LIN {X 116.112,Y 42.862,Z -30.023,A 90.000,B 90.000,C 0.000} C_DIS
LIN {X 115.370,Y 42.862,Z -29.775,A 90.000,B 90.000,C 0.000} C_DIS
LIN {X 114.612,Y 42.862,Z -29.581,A 90.000,B 90.000,C 0.000} C_DIS
LIN {X 113.842,Y 42.862,Z -29.441,A 90.000,B 90.000,C 0.000} C_DIS
LIN {X 113.064,Y 42.862,Z -29.357,A 90.000,B 90.000,C 0.000} C_DIS
LIN {X 112.897,Y 42.862,Z -29.321,A 90.000,B 90.000,C 0.000} C_DIS
LIN {X 111.921,Y 42.862,Z -29.250,A 90.000,B 90.000,C 0.000} C_DIS
LIN {X 110.943,Y 42.862,Z -29.245,A 90.000,B 90.000,C 0.000} C_DIS
LIN {X 109.967,Y 42.862,Z -29.306,A 90.000,B 90.000,C 0.000} C_DIS
LIN {X 108.997,Y 42.862,Z -29.432,A 90.000,B 90.000,C 0.000} C_DIS
LIN {X 108.037,Y 42.862,Z -29.624,A 90.000,B 90.000,C 0.000} C_DIS
LIN {X 107.093,Y 42.862,Z -29.879,A 90.000,B 90.000,C 0.000} C_DIS
LIN {X 106.168,Y 42.862,Z -30.198,A 90.000,B 90.000,C 0.000} C_DIS
LIN {X 105.267,Y 42.862,Z -30.578,A 90.000,B 90.000,C 0.000} C_DIS
LIN {X 104.393,Y 42.862,Z -31.018,A 90.000,B 90.000,C 0.000} C_DIS
LIN {X 103.550,Y 42.862,Z -31.515,A 90.000,B 90.000,C 0.000} C_DIS
LIN {X 102.744,Y 42.862,Z -32.069,A 90.000,B 90.000,C 0.000} C_DIS
LIN {X 101.486,Y 42.862,Z -33.150,A 90.000,B 90.000,C 0.000} C_DIS
LIN {X 100.261,Y 42.862,Z -34.268,A 90.000,B 90.000,C 0.000} C_DIS
LIN {X 99.071,Y 42.862,Z -35.423,A 90.000,B 90.000,C 0.000} C_DIS
LIN {X 97.915,Y 42.862,Z -36.613,A 90.000,B 90.000,C 0.000} C_DIS
LIN {X 96.796,Y 42.862,Z -37.837,A 90.000,B 90.000,C 0.000} C_DIS
LIN {X 95.769,Y 42.862,Z -39.072,A 90.000,B 90.000,C 0.000} C_DIS
LIN {X 94.703,Y 42.862,Z -40.275,A 90.000,B 90.000,C 0.000} C_DIS
LIN {X 93.600,Y 42.862,Z -41.444,A 90.000,B 90.000,C 0.000} C_DIS
LIN {X 92.461,Y 42.862,Z -42.577,A 90.000,B 90.000,C 0.000} C_DIS
LIN {X 91.287,Y 42.862,Z -43.675,A 90.000,B 90.000,C 0.000} C_DIS
LIN {X 90.080,Y 42.862,Z -44.735,A 90.000,B 90.000,C 0.000} C_DIS
LIN {X 88.132,Y 42.862,Z -46.382,A 90.000,B 90.000,C 0.000} C_DIS
LIN {X 86.196,Y 42.862,Z -48.042,A 90.000,B 90.000,C 0.000} C_DIS
LIN {X 84.951,Y 42.862,Z -49.069,A 90.000,B 90.000,C 0.000} C_DIS
LIN {X 83.746,Y 42.862,Z -50.143,A 90.000,B 90.000,C 0.000} C_DIS
LIN {X 82.582,Y 42.862,Z -51.262,A 90.000,B 90.000,C 0.000} C_DIS
LIN {X 81.462,Y 42.862,Z -52.424,A 90.000,B 90.000,C 0.000} C_DIS
LIN {X 80.387,Y 42.862,Z -53.629,A 90.000,B 90.000,C 0.000} C_DIS
LIN {X 79.359,Y 42.862,Z -54.873,A 90.000,B 90.000,C 0.000} C_DIS
LIN {X 78.378,Y 42.862,Z -56.155,A 90.000,B 90.000,C 0.000} C_DIS
LIN {X 77.447,Y 42.862,Z -57.474,A 90.000,B 90.000,C 0.000} C_DIS
LIN {X 76.567,Y 42.862,Z -58.827,A 90.000,B 90.000,C 0.000} C_DIS
LIN {X 75.739,Y 42.862,Z -60.212,A 90.000,B 90.000,C 0.000} C_DIS
LIN {X 74.965,Y 42.862,Z -61.629,A 90.000,B 90.000,C 0.000} C_DIS
LIN {X 74.244,Y 42.862,Z -63.073,A 90.000,B 90.000,C 0.000} C_DIS
LIN {X 73.845,Y 42.862,Z -63.813,A 90.000,B 90.000,C 0.000} C_DIS
LIN {X 73.487,Y 42.862,Z -64.573,A 90.000,B 90.000,C 0.000} C_DIS
LIN {X 73.171,Y 42.862,Z -65.351,A 90.000,B 90.000,C 0.000} C_DIS
LIN {X 72.898,Y 42.862,Z -66.146,A 90.000,B 90.000,C 0.000} C_DIS
LIN {X 72.667,Y 42.862,Z -66.954,A 90.000,B 90.000,C 0.000} C_DIS
LIN {X 72.481,Y 42.862,Z -67.773,A 90.000,B 90.000,C 0.000} C_DIS
LIN {X 72.193,Y 42.862,Z -67.636,A 90.000,B 90.000,C 0.000} C_DIS
LIN {X 71.927,Y 42.862,Z -67.460,A 90.000,B 90.000,C 0.000} C_DIS
LIN {X 71.688,Y 42.862,Z -67.248,A 90.000,B 90.000,C 0.000} C_DIS
LIN {X 71.483,Y 42.862,Z -67.004,A 90.000,B 90.000,C 0.000} C_DIS
LIN {X 71.429,Y 42.862,Z -66.954,A 90.000,B 90.000,C 0.000} C_DIS
LIN {X 70.953,Y 42.862,Z -66.449,A 90.000,B 90.000,C 0.000} C_DIS
LIN {X 70.447,Y 42.862,Z -65.973,A 90.000,B 90.000,C 0.000} C_DIS
LIN {X 69.914,Y 42.862,Z -65.529,A 90.000,B 90.000,C 0.000} C_DIS
LIN {X 69.429,Y 42.862,Z -64.681,A 90.000,B 90.000,C 0.000} C_DIS
LIN {X 68.963,Y 42.862,Z -63.823,A 90.000,B 90.000,C 0.000} C_DIS
LIN {X 68.514,Y 42.862,Z -62.956,A 90.000,B 90.000,C 0.000} C_DIS
LIN {X 68.048,Y 42.862,Z -61.606,A 90.000,B 90.000,C 0.000} C_DIS
LIN {X 67.516,Y 42.862,Z -60.281,A 90.000,B 90.000,C 0.000} C_DIS
LIN {X 66.919,Y 42.862,Z -58.984,A 90.000,B 90.000,C 0.000} C_DIS
LIN {X 66.258,Y 42.862,Z -57.718,A 90.000,B 90.000,C 0.000} C_DIS
LIN {X 65.535,Y 42.862,Z -56.486,A 90.000,B 90.000,C 0.000} C_DIS
LIN {X 64.753,Y 42.862,Z -55.292,A 90.000,B 90.000,C 0.000} C_DIS
LIN {X 63.912,Y 42.862,Z -54.138,A 90.000,B 90.000,C 0.000} C_DIS
LIN {X 63.016,Y 42.862,Z -53.026,A 90.000,B 90.000,C 0.000} C_DIS
LIN {X 62.065,Y 42.862,Z -51.961,A 90.000,B 90.000,C 0.000} C_DIS
LIN {X 61.384,Y 42.862,Z -51.162,A 90.000,B 90.000,C 0.000} C_DIS
LIN {X 60.653,Y 42.862,Z -50.408,A 90.000,B 90.000,C 0.000} C_DIS
LIN {X 59.875,Y 42.862,Z -49.703,A 90.000,B 90.000,C 0.000} C_DIS
LIN {X 59.052,Y 42.862,Z -49.049,A 90.000,B 90.000,C 0.000} C_DIS
LIN {X 58.190,Y 42.862,Z -48.450,A 90.000,B 90.000,C 0.000} C_DIS
LIN {X 57.290,Y 42.862,Z -47.908,A 90.000,B 90.000,C 0.000} C_DIS
LIN {X 56.358,Y 42.862,Z -47.426,A 90.000,B 90.000,C 0.000} C_DIS
LIN {X 55.396,Y 42.862,Z -47.004,A 90.000,B 90.000,C 0.000} C_DIS
LIN {X 54.409,Y 42.862,Z -46.645,A 90.000,B 90.000,C 0.000} C_DIS
LIN {X 53.401,Y 42.862,Z -46.351,A 90.000,B 90.000,C 0.000} C_DIS
LIN {X 52.526,Y 42.862,Z -46.091,A 90.000,B 90.000,C 0.000} C_DIS
LIN {X 51.636,Y 42.862,Z -45.891,A 90.000,B 90.000,C 0.000} C_DIS
LIN {X 50.735,Y 42.862,Z -45.751,A 90.000,B 90.000,C 0.000} C_DIS
LIN {X 49.826,Y 42.862,Z -45.672,A 90.000,B 90.000,C 0.000} C_DIS
LIN {X 48.914,Y 42.862,Z -45.655,A 90.000,B 90.000,C 0.000} C_DIS
LIN {X 48.002,Y 42.862,Z -45.698,A 90.000,B 90.000,C 0.000} C_DIS
LIN {X 47.096,Y 42.862,Z -45.803,A 90.000,B 90.000,C 0.000} C_DIS
LIN {X 46.154,Y 42.862,Z -45.305,A 90.000,B 90.000,C 0.000} C_DIS
LIN {X 45.179,Y 42.862,Z -44.876,A 90.000,B 90.000,C 0.000} C_DIS
LIN {X 44.175,Y 42.862,Z -44.518,A 90.000,B 90.000,C 0.000} C_DIS
LIN {X 43.148,Y 42.862,Z -44.234,A 90.000,B 90.000,C 0.000} C_DIS
LIN {X 42.104,Y 42.862,Z -44.025,A 90.000,B 90.000,C 0.000} C_DIS
LIN {X 41.046,Y 42.862,Z -43.892,A 90.000,B 90.000,C 0.000} C_DIS
LIN {X 39.983,Y 42.862,Z -43.835,A 90.000,B 90.000,C 0.000} C_DIS
LIN {X 38.917,Y 42.862,Z -43.855,A 90.000,B 90.000,C 0.000} C_DIS
LIN {X 37.856,Y 42.862,Z -43.953,A 90.000,B 90.000,C 0.000} C_DIS
LIN {X 36.805,Y 42.862,Z -44.126,A 90.000,B 90.000,C 0.000} C_DIS
LIN {X 35.769,Y 42.862,Z -44.375,A 90.000,B 90.000,C 0.000} C_DIS
LIN {X 34.754,Y 42.862,Z -44.698,A 90.000,B 90.000,C 0.000} C_DIS
LIN {X 33.764,Y 42.862,Z -45.093,A 90.000,B 90.000,C 0.000} C_DIS
LIN {X 32.806,Y 42.862,Z -45.559,A 90.000,B 90.000,C 0.000} C_DIS
LIN {X 31.884,Y 42.862,Z -46.093,A 90.000,B 90.000,C 0.000} C_DIS
LIN {X 31.003,Y 42.862,Z -46.692,A 90.000,B 90.000,C 0.000} C_DIS
LIN {X 30.167,Y 42.862,Z -47.353,A 90.000,B 90.000,C 0.000} C_DIS
LIN {X 29.381,Y 42.862,Z -48.073,A 90.000,B 90.000,C 0.000} C_DIS
LIN {X 28.650,Y 42.862,Z -48.847,A 90.000,B 90.000,C 0.000} C_DIS
LIN {X 27.976,Y 42.862,Z -49.672,A 90.000,B 90.000,C 0.000} C_DIS
LIN {X 27.363,Y 42.862,Z -50.544,A 90.000,B 90.000,C 0.000} C_DIS
LIN {X 26.815,Y 42.862,Z -51.458,A 90.000,B 90.000,C 0.000} C_DIS
LIN {X 26.334,Y 42.862,Z -52.409,A 90.000,B 90.000,C 0.000} C_DIS
LIN {X 25.923,Y 42.862,Z -53.392,A 90.000,B 90.000,C 0.000} C_DIS
LIN {X 25.585,Y 42.862,Z -54.402,A 90.000,B 90.000,C 0.000} C_DIS
LIN {X 25.045,Y 42.862,Z -54.903,A 90.000,B 90.000,C 0.000} C_DIS
LIN {X 24.535,Y 42.862,Z -55.436,A 90.000,B 90.000,C 0.000} C_DIS
LIN {X 24.057,Y 42.862,Z -55.997,A 90.000,B 90.000,C 0.000} C_DIS
LIN {X 23.613,Y 42.862,Z -56.585,A 90.000,B 90.000,C 0.000} C_DIS
LIN {X 23.205,Y 42.862,Z -57.199,A 90.000,B 90.000,C 0.000} C_DIS
LIN {X 22.794,Y 42.862,Z -58.043,A 90.000,B 90.000,C 0.000} C_DIS
LIN {X 22.437,Y 42.862,Z -58.911,A 90.000,B 90.000,C 0.000} C_DIS
LIN {X 22.137,Y 42.862,Z -59.800,A 90.000,B 90.000,C 0.000} C_DIS
LIN {X 21.893,Y 42.862,Z -60.706,A 90.000,B 90.000,C 0.000} C_DIS
LIN {X 21.708,Y 42.862,Z -61.626,A 90.000,B 90.000,C 0.000} C_DIS
LIN {X 21.582,Y 42.862,Z -62.556,A 90.000,B 90.000,C 0.000} C_DIS
LIN {X 21.515,Y 42.862,Z -63.492,A 90.000,B 90.000,C 0.000} C_DIS
LIN {X 20.626,Y 42.862,Z -63.513,A 90.000,B 90.000,C 0.000} C_DIS
LIN {X 19.742,Y 42.862,Z -63.600,A 90.000,B 90.000,C 0.000} C_DIS
LIN {X 18.866,Y 42.862,Z -63.754,A 90.000,B 90.000,C 0.000} C_DIS
LIN {X 18.004,Y 42.862,Z -63.973,A 90.000,B 90.000,C 0.000} C_DIS
LIN {X 17.162,Y 42.862,Z -64.256,A 90.000,B 90.000,C 0.000} C_DIS
LIN {X 16.343,Y 42.862,Z -64.602,A 90.000,B 90.000,C 0.000} C_DIS
LIN {X 15.598,Y 42.862,Z -64.971,A 90.000,B 90.000,C 0.000} C_DIS
LIN {X 14.887,Y 42.862,Z -65.404,A 90.000,B 90.000,C 0.000} C_DIS
LIN {X 14.216,Y 42.862,Z -65.895,A 90.000,B 90.000,C 0.000} C_DIS
LIN {X 13.591,Y 42.862,Z -66.443,A 90.000,B 90.000,C 0.000} C_DIS
LIN {X 13.014,Y 42.862,Z -67.043,A 90.000,B 90.000,C 0.000} C_DIS
LIN {X 12.491,Y 42.862,Z -67.690,A 90.000,B 90.000,C 0.000} C_DIS
LIN {X 12.026,Y 42.862,Z -68.379,A 90.000,B 90.000,C 0.000} C_DIS
LIN {X 11.622,Y 42.862,Z -69.106,A 90.000,B 90.000,C 0.000} C_DIS
LIN {X 11.282,Y 42.862,Z -69.865,A 90.000,B 90.000,C 0.000} C_DIS
LIN {X 11.009,Y 42.862,Z -70.651,A 90.000,B 90.000,C 0.000} C_DIS
LIN {X 10.804,Y 42.862,Z -71.457,A 90.000,B 90.000,C 0.000} C_DIS
LIN {X 10.670,Y 42.862,Z -72.278,A 90.000,B 90.000,C 0.000} C_DIS
LIN {X 10.606,Y 42.862,Z -73.107,A 90.000,B 90.000,C 0.000} C_DIS
LIN {X 10.606,Y 55.362,Z -73.107,A 90.000,B 90.000,C 0.000} C_DIS
LIN {X 10.606,Y 67.862,Z -73.107,A 90.000,B 90.000,C 0.000} C_DIS
LIN {X -110.439,Y 67.862,Z -242.561,A 90.000,B 90.000,C 0.000} C_DIS
LIN {X -110.439,Y 60.719,Z -242.561,A 90.000,B 90.000,C 0.000} C_DIS
LIN {X -110.439,Y 48.219,Z -242.561,A 90.000,B 90.000,C 0.000} C_DIS
LIN {X -110.439,Y 35.719,Z -242.561,A 90.000,B 90.000,C 0.000} C_DIS
LIN {X -144.015,Y 35.719,Z -242.561,A 90.000,B 90.000,C 0.000} C_DIS
LIN {X -144.015,Y 35.719,Z -235.012,A 90.000,B 90.000,C 0.000} C_DIS
LIN {X -100.322,Y 35.719,Z -235.012,A 90.000,B 90.000,C 0.000} C_DIS
LIN {X -97.556,Y 35.719,Z -233.079,A 90.000,B 90.000,C 0.000} C_DIS
LIN {X -94.768,Y 35.719,Z -231.176,A 90.000,B 90.000,C 0.000} C_DIS
LIN {X -91.960,Y 35.719,Z -229.305,A 90.000,B 90.000,C 0.000} C_DIS
LIN {X -89.131,Y 35.719,Z -227.464,A 90.000,B 90.000,C 0.000} C_DIS
LIN {X -144.015,Y 35.719,Z -227.464,A 90.000,B 90.000,C 0.000} C_DIS
LIN {X -144.015,Y 35.719,Z -219.915,A 90.000,B 90.000,C 0.000} C_DIS
LIN {X -76.760,Y 35.719,Z -219.915,A 90.000,B 90.000,C 0.000} C_DIS
LIN {X -73.331,Y 35.719,Z -217.961,A 90.000,B 90.000,C 0.000} C_DIS
LIN {X -69.877,Y 35.719,Z -216.051,A 90.000,B 90.000,C 0.000} C_DIS
LIN {X -66.399,Y 35.719,Z -214.186,A 90.000,B 90.000,C 0.000} C_DIS
LIN {X -62.897,Y 35.719,Z -212.366,A 90.000,B 90.000,C 0.000} C_DIS
LIN {X -144.015,Y 35.719,Z -212.366,A 90.000,B 90.000,C 0.000} C_DIS
LIN {X -144.015,Y 35.719,Z -204.817,A 90.000,B 90.000,C 0.000} C_DIS
LIN {X -47.547,Y 35.719,Z -204.817,A 90.000,B 90.000,C 0.000} C_DIS
LIN {X -47.331,Y 35.719,Z -204.710,A 90.000,B 90.000,C 0.000} C_DIS
LIN {X -44.561,Y 35.719,Z -203.328,A 90.000,B 90.000,C 0.000} C_DIS
LIN {X -41.819,Y 35.719,Z -201.892,A 90.000,B 90.000,C 0.000} C_DIS
LIN {X -39.105,Y 35.719,Z -200.403,A 90.000,B 90.000,C 0.000} C_DIS
LIN {X -36.421,Y 35.719,Z -198.862,A 90.000,B 90.000,C 0.000} C_DIS
LIN {X -33.767,Y 35.719,Z -197.269,A 90.000,B 90.000,C 0.000} C_DIS
LIN {X -144.015,Y 35.719,Z -197.269,A 90.000,B 90.000,C 0.000} C_DIS
LIN {X -144.015,Y 35.719,Z -189.720,A 90.000,B 90.000,C 0.000} C_DIS
LIN {X -22.669,Y 35.719,Z -189.720,A 90.000,B 90.000,C 0.000} C_DIS
LIN {X -20.312,Y 35.719,Z -187.881,A 90.000,B 90.000,C 0.000} C_DIS
LIN {X -17.981,Y 35.719,Z -186.010,A 90.000,B 90.000,C 0.000} C_DIS
LIN {X -15.676,Y 35.719,Z -184.106,A 90.000,B 90.000,C 0.000} C_DIS
LIN {X -13.397,Y 35.719,Z -182.171,A 90.000,B 90.000,C 0.000} C_DIS
LIN {X -144.015,Y 35.719,Z -182.171,A 90.000,B 90.000,C 0.000} C_DIS
LIN {X -144.015,Y 35.719,Z -174.622,A 90.000,B 90.000,C 0.000} C_DIS
LIN {X -5.086,Y 35.719,Z -174.622,A 90.000,B 90.000,C 0.000} C_DIS
LIN {X -3.303,Y 35.719,Z -172.895,A 90.000,B 90.000,C 0.000} C_DIS
LIN {X -1.540,Y 35.719,Z -171.148,A 90.000,B 90.000,C 0.000} C_DIS
LIN {X 0.203,Y 35.719,Z -169.380,A 90.000,B 90.000,C 0.000} C_DIS
LIN {X 0.708,Y 35.719,Z -168.847,A 90.000,B 90.000,C 0.000} C_DIS
LIN {X 1.178,Y 35.719,Z -168.284,A 90.000,B 90.000,C 0.000} C_DIS
LIN {X 1.612,Y 35.719,Z -167.691,A 90.000,B 90.000,C 0.000} C_DIS
LIN {X 2.008,Y 35.719,Z -167.073,A 90.000,B 90.000,C 0.000} C_DIS
LIN {X -144.015,Y 35.719,Z -167.073,A 90.000,B 90.000,C 0.000} C_DIS
LIN {X -144.015,Y 35.719,Z -159.525,A 90.000,B 90.000,C 0.000} C_DIS
LIN {X -13.056,Y 35.719,Z -159.525,A 90.000,B 90.000,C 0.000} C_DIS
LIN {X -14.940,Y 35.719,Z -158.616,A 90.000,B 90.000,C 0.000} C_DIS
LIN {X -16.795,Y 35.719,Z -157.649,A 90.000,B 90.000,C 0.000} C_DIS
LIN {X -18.619,Y 35.719,Z -156.624,A 90.000,B 90.000,C 0.000} C_DIS
LIN {X -20.410,Y 35.719,Z -155.544,A 90.000,B 90.000,C 0.000} C_DIS
LIN {X -22.167,Y 35.719,Z -154.408,A 90.000,B 90.000,C 0.000} C_DIS
LIN {X -23.888,Y 35.719,Z -153.219,A 90.000,B 90.000,C 0.000} C_DIS
LIN {X -25.571,Y 35.719,Z -151.976,A 90.000,B 90.000,C 0.000} C_DIS
LIN {X -144.015,Y 35.719,Z -151.976,A 90.000,B 90.000,C 0.000} C_DIS
LIN {X -144.015,Y 35.719,Z -144.427,A 90.000,B 90.000,C 0.000} C_DIS
LIN {X -34.283,Y 35.719,Z -144.427,A 90.000,B 90.000,C 0.000} C_DIS
LIN {X -35.276,Y 35.719,Z -143.415,A 90.000,B 90.000,C 0.000} C_DIS
LIN {X -36.235,Y 35.719,Z -142.372,A 90.000,B 90.000,C 0.000} C_DIS
LIN {X -37.160,Y 35.719,Z -141.298,A 90.000,B 90.000,C 0.000} C_DIS
LIN {X -38.050,Y 35.719,Z -140.194,A 90.000,B 90.000,C 0.000} C_DIS
LIN {X -38.903,Y 35.719,Z -139.062,A 90.000,B 90.000,C 0.000} C_DIS
LIN {X -39.719,Y 35.719,Z -137.903,A 90.000,B 90.000,C 0.000} C_DIS
LIN {X -40.068,Y 35.719,Z -137.393,A 90.000,B 90.000,C 0.000} C_DIS
LIN {X -40.411,Y 35.719,Z -136.878,A 90.000,B 90.000,C 0.000} C_DIS
LIN {X -144.015,Y 35.719,Z -136.878,A 90.000,B 90.000,C 0.000} C_DIS
LIN {X -144.015,Y 35.719,Z -129.329,A 90.000,B 90.000,C 0.000} C_DIS
LIN {X -44.482,Y 35.719,Z -129.329,A 90.000,B 90.000,C 0.000} C_DIS
LIN {X -45.091,Y 35.719,Z -127.854,A 90.000,B 90.000,C 0.000} C_DIS
LIN {X -45.652,Y 35.719,Z -126.360,A 90.000,B 90.000,C 0.000} C_DIS
LIN {X -46.164,Y 35.719,Z -124.849,A 90.000,B 90.000,C 0.000} C_DIS
LIN {X -46.628,Y 35.719,Z -123.322,A 90.000,B 90.000,C 0.000} C_DIS
LIN {X -47.042,Y 35.719,Z -121.781,A 90.000,B 90.000,C 0.000} C_DIS
LIN {X -144.015,Y 35.719,Z -121.781,A 90.000,B 90.000,C 0.000} C_DIS
LIN {X -144.015,Y 35.719,Z -114.232,A 90.000,B 90.000,C 0.000} C_DIS
LIN {X -48.326,Y 35.719,Z -114.232,A 90.000,B 90.000,C 0.000} C_DIS
LIN {X -48.439,Y 35.719,Z -112.740,A 90.000,B 90.000,C 0.000} C_DIS
LIN {X -48.508,Y 35.719,Z -111.245,A 90.000,B 90.000,C 0.000} C_DIS
LIN {X -48.531,Y 35.719,Z -109.749,A 90.000,B 90.000,C 0.000} C_DIS
LIN {X -49.255,Y 35.719,Z -108.705,A 90.000,B 90.000,C 0.000} C_DIS
LIN {X -50.009,Y 35.719,Z -107.683,A 90.000,B 90.000,C 0.000} C_DIS
LIN {X -50.793,Y 35.719,Z -106.683,A 90.000,B 90.000,C 0.000} C_DIS
LIN {X -144.015,Y 35.719,Z -106.683,A 90.000,B 90.000,C 0.000} C_DIS
LIN {X -144.015,Y 35.719,Z -99.134,A 90.000,B 90.000,C 0.000} C_DIS
LIN {X -55.690,Y 35.719,Z -99.134,A 90.000,B 90.000,C 0.000} C_DIS
LIN {X -56.171,Y 35.719,Z -98.249,A 90.000,B 90.000,C 0.000} C_DIS
LIN {X -56.638,Y 35.719,Z -97.357,A 90.000,B 90.000,C 0.000} C_DIS
LIN {X -57.300,Y 35.719,Z -95.943,A 90.000,B 90.000,C 0.000} C_DIS
LIN {X -57.917,Y 35.719,Z -94.509,A 90.000,B 90.000,C 0.000} C_DIS
LIN {X -58.488,Y 35.719,Z -93.056,A 90.000,B 90.000,C 0.000} C_DIS
LIN {X -59.012,Y 35.719,Z -91.586,A 90.000,B 90.000,C 0.000} C_DIS
LIN {X -144.015,Y 35.719,Z -91.586,A 90.000,B 90.000,C 0.000} C_DIS
LIN {X -144.015,Y 35.719,Z -84.037,A 90.000,B 90.000,C 0.000} C_DIS
LIN {X -60.912,Y 35.719,Z -84.037,A 90.000,B 90.000,C 0.000} C_DIS
LIN {X -61.009,Y 35.719,Z -83.435,A 90.000,B 90.000,C 0.000} C_DIS
LIN {X -61.219,Y 35.719,Z -82.056,A 90.000,B 90.000,C 0.000} C_DIS
LIN {X -61.375,Y 35.719,Z -80.669,A 90.000,B 90.000,C 0.000} C_DIS
LIN {X -61.478,Y 35.719,Z -79.278,A 90.000,B 90.000,C 0.000} C_DIS
LIN {X -61.527,Y 35.719,Z -77.883,A 90.000,B 90.000,C 0.000} C_DIS
LIN {X -61.523,Y 35.719,Z -76.488,A 90.000,B 90.000,C 0.000} C_DIS
LIN {X -144.015,Y 35.719,Z -76.488,A 90.000,B 90.000,C 0.000} C_DIS
LIN {X -144.015,Y 35.719,Z -68.939,A 90.000,B 90.000,C 0.000} C_DIS
LIN {X -60.555,Y 35.719,Z -68.939,A 90.000,B 90.000,C 0.000} C_DIS
LIN {X -60.426,Y 35.719,Z -68.411,A 90.000,B 90.000,C 0.000} C_DIS
LIN {X -60.288,Y 35.719,Z -67.885,A 90.000,B 90.000,C 0.000} C_DIS
LIN {X -59.940,Y 35.719,Z -66.870,A 90.000,B 90.000,C 0.000} C_DIS
LIN {X -59.531,Y 35.719,Z -65.877,A 90.000,B 90.000,C 0.000} C_DIS
LIN {X -59.062,Y 35.719,Z -64.912,A 90.000,B 90.000,C 0.000} C_DIS
LIN {X -58.534,Y 35.719,Z -63.977,A 90.000,B 90.000,C 0.000} C_DIS
LIN {X -57.951,Y 35.719,Z -63.077,A 90.000,B 90.000,C 0.000} C_DIS
LIN {X -57.313,Y 35.719,Z -62.213,A 90.000,B 90.000,C 0.000} C_DIS
LIN {X -56.624,Y 35.719,Z -61.390,A 90.000,B 90.000,C 0.000} C_DIS
LIN {X -144.015,Y 35.719,Z -61.390,A 90.000,B 90.000,C 0.000} C_DIS
LIN {X -144.015,Y 35.719,Z -53.842,A 90.000,B 90.000,C 0.000} C_DIS
LIN {X -22.915,Y 35.719,Z -53.842,A 90.000,B 90.000,C 0.000} C_DIS
LIN {X -22.620,Y 35.719,Z -53.702,A 90.000,B 90.000,C 0.000} C_DIS
LIN {X -22.321,Y 35.719,Z -53.571,A 90.000,B 90.000,C 0.000} C_DIS
LIN {X -21.316,Y 35.719,Z -53.112,A 90.000,B 90.000,C 0.000} C_DIS
LIN {X -20.286,Y 35.719,Z -52.714,A 90.000,B 90.000,C 0.000} C_DIS
LIN {X -19.234,Y 35.719,Z -52.379,A 90.000,B 90.000,C 0.000} C_DIS
LIN {X -18.163,Y 35.719,Z -52.107,A 90.000,B 90.000,C 0.000} C_DIS
LIN {X -17.078,Y 35.719,Z -51.900,A 90.000,B 90.000,C 0.000} C_DIS
LIN {X -15.982,Y 35.719,Z -51.759,A 90.000,B 90.000,C 0.000} C_DIS
LIN {X -14.880,Y 35.719,Z -51.684,A 90.000,B 90.000,C 0.000} C_DIS
LIN {X -13.776,Y 35.719,Z -51.675,A 90.000,B 90.000,C 0.000} C_DIS
LIN {X -12.673,Y 35.719,Z -51.733,A 90.000,B 90.000,C 0.000} C_DIS
LIN {X -11.631,Y 35.719,Z -51.728,A 90.000,B 90.000,C 0.000} C_DIS
LIN {X -10.589,Y 35.719,Z -51.767,A 90.000,B 90.000,C 0.000} C_DIS
LIN {X 21.929,Y 35.719,Z -46.293,A 90.000,B 90.000,C 0.000} C_DIS
LIN {X -144.015,Y 35.719,Z -46.293,A 90.000,B 90.000,C 0.000} C_DIS
LIN {X -144.015,Y 35.719,Z -38.744,A 90.000,B 90.000,C 0.000} C_DIS
LIN {X 30.518,Y 35.719,Z -38.744,A 90.000,B 90.000,C 0.000} C_DIS
LIN {X 31.463,Y 35.719,Z -38.438,A 90.000,B 90.000,C 0.000} C_DIS
LIN {X 32.425,Y 35.719,Z -38.189,A 90.000,B 90.000,C 0.000} C_DIS
LIN {X 33.399,Y 35.719,Z -37.996,A 90.000,B 90.000,C 0.000} C_DIS
LIN {X 34.384,Y 35.719,Z -37.862,A 90.000,B 90.000,C 0.000} C_DIS
LIN {X 35.374,Y 35.719,Z -37.786,A 90.000,B 90.000,C 0.000} C_DIS
LIN {X 36.367,Y 35.719,Z -37.768,A 90.000,B 90.000,C 0.000} C_DIS
LIN {X 37.360,Y 35.719,Z -37.809,A 90.000,B 90.000,C 0.000} C_DIS
LIN {X 38.348,Y 35.719,Z -37.909,A 90.000,B 90.000,C 0.000} C_DIS
LIN {X 39.329,Y 35.719,Z -38.066,A 90.000,B 90.000,C 0.000} C_DIS
LIN {X 39.892,Y 35.719,Z -38.197,A 90.000,B 90.000,C 0.000} C_DIS
LIN {X 40.465,Y 35.719,Z -38.264,A 90.000,B 90.000,C 0.000} C_DIS
LIN {X 41.043,Y 35.719,Z -38.268,A 90.000,B 90.000,C 0.000} C_DIS
LIN {X 41.617,Y 35.719,Z -38.208,A 90.000,B 90.000,C 0.000} C_DIS
LIN {X 42.182,Y 35.719,Z -38.085,A 90.000,B 90.000,C 0.000} C_DIS
LIN {X 42.729,Y 35.719,Z -37.900,A 90.000,B 90.000,C 0.000} C_DIS
LIN {X 43.847,Y 35.719,Z -37.642,A 90.000,B 90.000,C 0.000} C_DIS
LIN {X 44.979,Y 35.719,Z -37.448,A 90.000,B 90.000,C 0.000} C_DIS
LIN {X 46.119,Y 35.719,Z -37.317,A 90.000,B 90.000,C 0.000} C_DIS
LIN {X 47.265,Y 35.719,Z -37.251,A 90.000,B 90.000,C 0.000} C_DIS
LIN {X 48.412,Y 35.719,Z -37.249,A 90.000,B 90.000,C 0.000} C_DIS
LIN {X 49.558,Y 35.719,Z -37.312,A 90.000,B 90.000,C 0.000} C_DIS
LIN {X 50.699,Y 35.719,Z -37.439,A 90.000,B 90.000,C 0.000} C_DIS
LIN {X 50.893,Y 35.719,Z -37.468,A 90.000,B 90.000,C 0.000} C_DIS
LIN {X 51.988,Y 35.719,Z -37.716,A 90.000,B 90.000,C 0.000} C_DIS
LIN {X 53.070,Y 35.719,Z -38.012,A 90.000,B 90.000,C 0.000} C_DIS
LIN {X 54.139,Y 35.719,Z -38.355,A 90.000,B 90.000,C 0.000} C_DIS
LIN {X 55.192,Y 35.719,Z -38.744,A 90.000,B 90.000,C 0.000} C_DIS
LIN {X 87.785,Y 35.719,Z -38.744,A 90.000,B 90.000,C 0.000} C_DIS
LIN {X 87.273,Y 35.719,Z -39.488,A 90.000,B 90.000,C 0.000} C_DIS
LIN {X 86.809,Y 35.719,Z -40.262,A 90.000,B 90.000,C 0.000} C_DIS
LIN {X 86.394,Y 35.719,Z -41.064,A 90.000,B 90.000,C 0.000} C_DIS
LIN {X 86.030,Y 35.719,Z -41.890,A 90.000,B 90.000,C 0.000} C_DIS
LIN {X 85.719,Y 35.719,Z -42.738,A 90.000,B 90.000,C 0.000} C_DIS
LIN {X 85.461,Y 35.719,Z -43.603,A 90.000,B 90.000,C 0.000} C_DIS
LIN {X 85.258,Y 35.719,Z -44.483,A 90.000,B 90.000,C 0.000} C_DIS
LIN {X 85.111,Y 35.719,Z -45.374,A 90.000,B 90.000,C 0.000} C_DIS
LIN {X 85.036,Y 35.719,Z -45.832,A 90.000,B 90.000,C 0.000} C_DIS
LIN {X 84.988,Y 35.719,Z -46.293,A 90.000,B 90.000,C 0.000} C_DIS
LIN {X 66.072,Y 35.719,Z -46.293,A 90.000,B 90.000,C 0.000} C_DIS
LIN {X 67.903,Y 35.719,Z -47.977,A 90.000,B 90.000,C 0.000} C_DIS
LIN {X 69.708,Y 35.719,Z -49.688,A 90.000,B 90.000,C 0.000} C_DIS
LIN {X 71.272,Y 35.719,Z -51.045,A 90.000,B 90.000,C 0.000} C_DIS
LIN {X 72.812,Y 35.719,Z -52.430,A 90.000,B 90.000,C 0.000} C_DIS
LIN {X 74.327,Y 35.719,Z -53.842,A 90.000,B 90.000,C 0.000} C_DIS
LIN {X 78.925,Y 35.719,Z -53.842,A 90.000,B 90.000,C 0.000} C_DIS
LIN {X 79.855,Y 35.719,Z -52.742,A 90.000,B 90.000,C 0.000} C_DIS
LIN {X 80.820,Y 35.719,Z -51.673,A 90.000,B 90.000,C 0.000} C_DIS
LIN {X 81.819,Y 35.719,Z -50.635,A 90.000,B 90.000,C 0.000} C_DIS
LIN {X 82.851,Y 35.719,Z -49.631,A 90.000,B 90.000,C 0.000} C_DIS
LIN {X 83.916,Y 35.719,Z -48.660,A 90.000,B 90.000,C 0.000} C_DIS
LIN {X 85.010,Y 35.719,Z -47.724,A 90.000,B 90.000,C 0.000} C_DIS
LIN {X 84.969,Y 35.719,Z -47.135,A 90.000,B 90.000,C 0.000} C_DIS
LIN {X 84.973,Y 35.719,Z -46.545,A 90.000,B 90.000,C 0.000} C_DIS
LIN {X 85.020,Y 35.719,Z -45.957,A 90.000,B 90.000,C 0.000} C_DIS
LIN {X 85.111,Y 35.719,Z -45.374,A 90.000,B 90.000,C 0.000} C_DIS
LIN {X 85.265,Y 35.719,Z -44.448,A 90.000,B 90.000,C 0.000} C_DIS
LIN {X 85.479,Y 35.719,Z -43.535,A 90.000,B 90.000,C 0.000} C_DIS
LIN {X 85.752,Y 35.719,Z -42.637,A 90.000,B 90.000,C 0.000} C_DIS
LIN {X 86.084,Y 35.719,Z -41.759,A 90.000,B 90.000,C 0.000} C_DIS
LIN {X 86.471,Y 35.719,Z -40.904,A 90.000,B 90.000,C 0.000} C_DIS
LIN {X 86.914,Y 35.719,Z -40.077,A 90.000,B 90.000,C 0.000} C_DIS
LIN {X 87.409,Y 35.719,Z -39.280,A 90.000,B 90.000,C 0.000} C_DIS
LIN {X 87.955,Y 35.719,Z -38.517,A 90.000,B 90.000,C 0.000} C_DIS
LIN {X 88.550,Y 35.719,Z -37.791,A 90.000,B 90.000,C 0.000} C_DIS
LIN {X 89.261,Y 35.719,Z -36.989,A 90.000,B 90.000,C 0.000} C_DIS
LIN {X 90.014,Y 35.719,Z -36.226,A 90.000,B 90.000,C 0.000} C_DIS
LIN {X 90.806,Y 35.719,Z -35.505,A 90.000,B 90.000,C 0.000} C_DIS
LIN {X 91.636,Y 35.719,Z -34.827,A 90.000,B 90.000,C 0.000} C_DIS
LIN {X 92.502,Y 35.719,Z -34.195,A 90.000,B 90.000,C 0.000} C_DIS
LIN {X 93.400,Y 35.719,Z -33.610,A 90.000,B 90.000,C 0.000} C_DIS
LIN {X 94.327,Y 35.719,Z -33.074,A 90.000,B 90.000,C 0.000} C_DIS
LIN {X 95.283,Y 35.719,Z -32.588,A 90.000,B 90.000,C 0.000} C_DIS
LIN {X 96.263,Y 35.719,Z -32.155,A 90.000,B 90.000,C 0.000} C_DIS
LIN {X 98.348,Y 35.719,Z -31.177,A 90.000,B 90.000,C 0.000} C_DIS
LIN {X 100.456,Y 35.719,Z -30.251,A 90.000,B 90.000,C 0.000} C_DIS
LIN {X 102.587,Y 35.719,Z -29.378,A 90.000,B 90.000,C 0.000} C_DIS
LIN {X 104.739,Y 35.719,Z -28.558,A 90.000,B 90.000,C 0.000} C_DIS
LIN {X 106.910,Y 35.719,Z -27.791,A 90.000,B 90.000,C 0.000} C_DIS
LIN {X 107.872,Y 35.719,Z -27.586,A 90.000,B 90.000,C 0.000} C_DIS
LIN {X 108.844,Y 35.719,Z -27.444,A 90.000,B 90.000,C 0.000} C_DIS
LIN {X 109.825,Y 35.719,Z -27.367,A 90.000,B 90.000,C 0.000} C_DIS
LIN {X 110.808,Y 35.719,Z -27.353,A 90.000,B 90.000,C 0.000} C_DIS
LIN {X 111.789,Y 35.719,Z -27.403,A 90.000,B 90.000,C 0.000} C_DIS
LIN {X 112.766,Y 35.719,Z -27.518,A 90.000,B 90.000,C 0.000} C_DIS
LIN {X 113.733,Y 35.719,Z -27.696,A 90.000,B 90.000,C 0.000} C_DIS
LIN {X 114.686,Y 35.719,Z -27.937,A 90.000,B 90.000,C 0.000} C_DIS
LIN {X 114.871,Y 35.719,Z -27.996,A 90.000,B 90.000,C 0.000} C_DIS
LIN {X 115.775,Y 35.719,Z -28.294,A 90.000,B 90.000,C 0.000} C_DIS
LIN {X 116.659,Y 35.719,Z -28.648,A 90.000,B 90.000,C 0.000} C_DIS
LIN {X 117.519,Y 35.719,Z -29.056,A 90.000,B 90.000,C 0.000} C_DIS
LIN {X 118.352,Y 35.719,Z -29.518,A 90.000,B 90.000,C 0.000} C_DIS
LIN {X 118.488,Y 35.719,Z -29.602,A 90.000,B 90.000,C 0.000} C_DIS
LIN {X 119.051,Y 35.719,Z -29.962,A 90.000,B 90.000,C 0.000} C_DIS
LIN {X 119.596,Y 35.719,Z -30.349,A 90.000,B 90.000,C 0.000} C_DIS
LIN {X 120.122,Y 35.719,Z -30.760,A 90.000,B 90.000,C 0.000} C_DIS
LIN {X 120.629,Y 35.719,Z -31.195,A 90.000,B 90.000,C 0.000} C_DIS
LIN {X 144.015,Y 35.719,Z -31.195,A 90.000,B 90.000,C 0.000} C_DIS
LIN {X 144.015,Y 35.719,Z -38.744,A 90.000,B 90.000,C 0.000} C_DIS
LIN {X 125.014,Y 35.719,Z -38.744,A 90.000,B 90.000,C 0.000} C_DIS
LIN {X 125.231,Y 35.719,Z -39.809,A 90.000,B 90.000,C 0.000} C_DIS
LIN {X 125.383,Y 35.719,Z -40.885,A 90.000,B 90.000,C 0.000} C_DIS
LIN {X 125.467,Y 35.719,Z -41.969,A 90.000,B 90.000,C 0.000} C_DIS
LIN {X 125.484,Y 35.719,Z -43.056,A 90.000,B 90.000,C 0.000} C_DIS
LIN {X 125.434,Y 35.719,Z -44.141,A 90.000,B 90.000,C 0.000} C_DIS
LIN {X 125.317,Y 35.719,Z -45.222,A 90.000,B 90.000,C 0.000} C_DIS
LIN {X 125.133,Y 35.719,Z -46.293,A 90.000,B 90.000,C 0.000} C_DIS
LIN {X 144.015,Y 35.719,Z -46.293,A 90.000,B 90.000,C 0.000} C_DIS
LIN {X 144.015,Y 35.719,Z -53.842,A 90.000,B 90.000,C 0.000} C_DIS
LIN {X 122.348,Y 35.719,Z -53.842,A 90.000,B 90.000,C 0.000} C_DIS
LIN {X 122.049,Y 35.719,Z -54.392,A 90.000,B 90.000,C 0.000} C_DIS
LIN {X 121.738,Y 35.719,Z -54.936,A 90.000,B 90.000,C 0.000} C_DIS
LIN {X 121.121,Y 35.719,Z -56.194,A 90.000,B 90.000,C 0.000} C_DIS
LIN {X 120.541,Y 35.719,Z -57.469,A 90.000,B 90.000,C 0.000} C_DIS
LIN {X 119.999,Y 35.719,Z -58.761,A 90.000,B 90.000,C 0.000} C_DIS
LIN {X 119.494,Y 35.719,Z -60.068,A 90.000,B 90.000,C 0.000} C_DIS
LIN {X 119.029,Y 35.719,Z -61.390,A 90.000,B 90.000,C 0.000} C_DIS
LIN {X 144.015,Y 35.719,Z -61.390,A 90.000,B 90.000,C 0.000} C_DIS
LIN {X 144.015,Y 35.719,Z -68.939,A 90.000,B 90.000,C 0.000} C_DIS
LIN {X 116.890,Y 35.719,Z -68.939,A 90.000,B 90.000,C 0.000} C_DIS
LIN {X 116.236,Y 35.719,Z -70.854,A 90.000,B 90.000,C 0.000} C_DIS
LIN {X 115.533,Y 35.719,Z -72.752,A 90.000,B 90.000,C 0.000} C_DIS
LIN {X 114.781,Y 35.719,Z -74.630,A 90.000,B 90.000,C 0.000} C_DIS
LIN {X 113.979,Y 35.719,Z -76.488,A 90.000,B 90.000,C 0.000} C_DIS
LIN {X 144.015,Y 35.719,Z -76.488,A 90.000,B 90.000,C 0.000} C_DIS
LIN {X 144.015,Y 35.719,Z -84.037,A 90.000,B 90.000,C 0.000} C_DIS
LIN {X 110.099,Y 35.719,Z -84.037,A 90.000,B 90.000,C 0.000} C_DIS
LIN {X 109.231,Y 35.719,Z -85.483,A 90.000,B 90.000,C 0.000} C_DIS
LIN {X 108.332,Y 35.719,Z -86.910,A 90.000,B 90.000,C 0.000} C_DIS
LIN {X 107.403,Y 35.719,Z -88.318,A 90.000,B 90.000,C 0.000} C_DIS
LIN {X 106.442,Y 35.719,Z -89.704,A 90.000,B 90.000,C 0.000} C_DIS
LIN {X 106.288,Y 35.719,Z -91.586,A 90.000,B 90.000,C 0.000} C_DIS
LIN {X 144.015,Y 35.719,Z -91.586,A 90.000,B 90.000,C 0.000} C_DIS
LIN {X 144.015,Y 35.719,Z -99.134,A 90.000,B 90.000,C 0.000} C_DIS
LIN {X 105.272,Y 35.719,Z -99.134,A 90.000,B 90.000,C 0.000} C_DIS
LIN {X 104.934,Y 35.719,Z -100.380,A 90.000,B 90.000,C 0.000} C_DIS
LIN {X 104.562,Y 35.719,Z -101.616,A 90.000,B 90.000,C 0.000} C_DIS
LIN {X 104.157,Y 35.719,Z -102.842,A 90.000,B 90.000,C 0.000} C_DIS
LIN {X 103.885,Y 35.719,Z -103.883,A 90.000,B 90.000,C 0.000} C_DIS
LIN {X 103.655,Y 35.719,Z -104.934,A 90.000,B 90.000,C 0.000} C_DIS
LIN {X 103.774,Y 35.719,Z -105.808,A 90.000,B 90.000,C 0.000} C_DIS
LIN {X 103.879,Y 35.719,Z -106.683,A 90.000,B 90.000,C 0.000} C_DIS
LIN {X 144.015,Y 35.719,Z -106.683,A 90.000,B 90.000,C 0.000} C_DIS
LIN {X 144.015,Y 35.719,Z -114.232,A 90.000,B 90.000,C 0.000} C_DIS
LIN {X 104.169,Y 35.719,Z -114.232,A 90.000,B 90.000,C 0.000} C_DIS
LIN {X 104.141,Y 35.719,Z -114.921,A 90.000,B 90.000,C 0.000} C_DIS
LIN {X 104.185,Y 35.719,Z -117.555,A 90.000,B 90.000,C 0.000} C_DIS
LIN {X 104.247,Y 35.719,Z -120.189,A 90.000,B 90.000,C 0.000} C_DIS
LIN {X 104.266,Y 35.719,Z -120.985,A 90.000,B 90.000,C 0.000} C_DIS
LIN {X 104.278,Y 35.719,Z -121.781,A 90.000,B 90.000,C 0.000} C_DIS
LIN {X 144.015,Y 35.719,Z -121.781,A 90.000,B 90.000,C 0.000} C_DIS
LIN {X 144.015,Y 35.719,Z -129.329,A 90.000,B 90.000,C 0.000} C_DIS
LIN {X 104.096,Y 35.719,Z -129.329,A 90.000,B 90.000,C 0.000} C_DIS
LIN {X 103.960,Y 35.719,Z -131.270,A 90.000,B 90.000,C 0.000} C_DIS
LIN {X 103.788,Y 35.719,Z -133.209,A 90.000,B 90.000,C 0.000} C_DIS
LIN {X 103.580,Y 35.719,Z -135.144,A 90.000,B 90.000,C 0.000} C_DIS
LIN {X 103.443,Y 35.719,Z -136.878,A 90.000,B 90.000,C 0.000} C_DIS
LIN {X 144.015,Y 35.719,Z -136.878,A 90.000,B 90.000,C 0.000} C_DIS
LIN {X 144.015,Y 35.719,Z -144.427,A 90.000,B 90.000,C 0.000} C_DIS
LIN {X 102.703,Y 35.719,Z -144.427,A 90.000,B 90.000,C 0.000} C_DIS
LIN {X 102.404,Y 35.719,Z -146.947,A 90.000,B 90.000,C 0.000} C_DIS
LIN {X 102.078,Y 35.719,Z -149.463,A 90.000,B 90.000,C 0.000} C_DIS
LIN {X 101.726,Y 35.719,Z -151.976,A 90.000,B 90.000,C 0.000} C_DIS
LIN {X 144.015,Y 35.719,Z -151.976,A 90.000,B 90.000,C 0.000} C_DIS
LIN {X 144.015,Y 35.719,Z -159.525,A 90.000,B 90.000,C 0.000} C_DIS
LIN {X 100.462,Y 35.719,Z -159.525,A 90.000,B 90.000,C 0.000} C_DIS
LIN {X 99.903,Y 35.719,Z -162.050,A 90.000,B 90.000,C 0.000} C_DIS
LIN {X 99.304,Y 35.719,Z -164.567,A 90.000,B 90.000,C 0.000} C_DIS
LIN {X 98.666,Y 35.719,Z -167.073,A 90.000,B 90.000,C 0.000} C_DIS
LIN {X 144.015,Y 35.719,Z -167.073,A 90.000,B 90.000,C 0.000} C_DIS
LIN {X 144.015,Y 35.719,Z -174.622,A 90.000,B 90.000,C 0.000} C_DIS
LIN {X 96.486,Y 35.719,Z -174.622,A 90.000,B 90.000,C 0.000} C_DIS
LIN {X 96.025,Y 35.719,Z -176.063,A 90.000,B 90.000,C 0.000} C_DIS
LIN {X 95.550,Y 35.719,Z -177.500,A 90.000,B 90.000,C 0.000} C_DIS
LIN {X 94.065,Y 35.719,Z -182.171,A 90.000,B 90.000,C 0.000} C_DIS
LIN {X 144.015,Y 35.719,Z -182.171,A 90.000,B 90.000,C 0.000} C_DIS
LIN {X 144.015,Y 35.719,Z -189.720,A 90.000,B 90.000,C 0.000} C_DIS
LIN {X 91.678,Y 35.719,Z -189.720,A 90.000,B 90.000,C 0.000} C_DIS
LIN {X 90.456,Y 35.719,Z -193.500,A 90.000,B 90.000,C 0.000} C_DIS
LIN {X 89.200,Y 35.719,Z -197.269,A 90.000,B 90.000,C 0.000} C_DIS
LIN {X 144.015,Y 35.719,Z -197.269,A 90.000,B 90.000,C 0.000} C_DIS
LIN {X 144.015,Y 35.719,Z -204.817,A 90.000,B 90.000,C 0.000} C_DIS
LIN {X 86.571,Y 35.719,Z -204.817,A 90.000,B 90.000,C 0.000} C_DIS
LIN {X 85.196,Y 35.719,Z -208.598,A 90.000,B 90.000,C 0.000} C_DIS
LIN {X 83.787,Y 35.719,Z -212.366,A 90.000,B 90.000,C 0.000} C_DIS
LIN {X 144.015,Y 35.719,Z -212.366,A 90.000,B 90.000,C 0.000} C_DIS
LIN {X 144.015,Y 35.719,Z -219.915,A 90.000,B 90.000,C 0.000} C_DIS
LIN {X 80.845,Y 35.719,Z -219.915,A 90.000,B 90.000,C 0.000} C_DIS
LIN {X 79.311,Y 35.719,Z -223.697,A 90.000,B 90.000,C 0.000} C_DIS
LIN {X 77.743,Y 35.719,Z -227.464,A 90.000,B 90.000,C 0.000} C_DIS
LIN {X 144.015,Y 35.719,Z -227.464,A 90.000,B 90.000,C 0.000} C_DIS
LIN {X 144.015,Y 35.719,Z -235.012,A 90.000,B 90.000,C 0.000} C_DIS
LIN {X 74.495,Y 35.719,Z -235.012,A 90.000,B 90.000,C 0.000} C_DIS
LIN {X 73.727,Y 35.719,Z -236.918,A 90.000,B 90.000,C 0.000} C_DIS
LIN {X 72.919,Y 35.719,Z -238.807,A 90.000,B 90.000,C 0.000} C_DIS
LIN {X 71.415,Y 35.719,Z -242.561,A 90.000,B 90.000,C 0.000} C_DIS
LIN {X 144.015,Y 35.719,Z -242.561,A 90.000,B 90.000,C 0.000} C_DIS
LIN {X 144.015,Y 35.719,Z -23.646,A 90.000,B 90.000,C 0.000} C_DIS
LIN {X -144.015,Y 35.719,Z -23.646,A 90.000,B 90.000,C 0.000} C_DIS
LIN {X -144.015,Y 35.719,Z -16.098,A 90.000,B 90.000,C 0.000} C_DIS
LIN {X 144.015,Y 35.719,Z -16.098,A 90.000,B 90.000,C 0.000} C_DIS
LIN {X 144.015,Y 35.719,Z -8.549,A 90.000,B 90.000,C 0.000} C_DIS
LIN {X -144.015,Y 35.719,Z -8.549,A 90.000,B 90.000,C 0.000} C_DIS
LIN {X -144.015,Y 35.719,Z -1.000,A 90.000,B 90.000,C 0.000} C_DIS
LIN {X 144.015,Y 35.719,Z -1.000,A 90.000,B 90.000,C 0.000} C_DIS
LIN {X 98.307,Y 35.719,Z -31.195,A 90.000,B 90.000,C 0.000} C_DIS
LIN {X -144.015,Y 35.719,Z -31.195,A 90.000,B 90.000,C 0.000} C_DIS
LIN {X 5.050,Y 35.719,Z -53.842,A 90.000,B 90.000,C 0.000} C_DIS
LIN {X 9.338,Y 35.719,Z -53.842,A 90.000,B 90.000,C 0.000} C_DIS
LIN {X 9.139,Y 35.719,Z -55.051,A 90.000,B 90.000,C 0.000} C_DIS
LIN {X 7.500,Y 35.719,Z -55.000,A 90.000,B 90.000,C 0.000} C_DIS
LIN {X 5.862,Y 35.719,Z -54.907,A 90.000,B 90.000,C 0.000} C_DIS
LIN {X 4.227,Y 35.719,Z -54.772,A 90.000,B 90.000,C 0.000} C_DIS
LIN {X 2.597,Y 35.719,Z -54.594,A 90.000,B 90.000,C 0.000} C_DIS
LIN {X -2.801,Y 35.719,Z -53.794,A 90.000,B 90.000,C 0.000} C_DIS
LIN {X -8.205,Y 35.719,Z -53.038,A 90.000,B 90.000,C 0.000} C_DIS
LIN {X -9.322,Y 35.719,Z -52.881,A 90.000,B 90.000,C 0.000} C_DIS
LIN {X -10.446,Y 35.719,Z -52.778,A 90.000,B 90.000,C 0.000} C_DIS
LIN {X -11.573,Y 35.719,Z -52.728,A 90.000,B 90.000,C 0.000} C_DIS
LIN {X -12.701,Y 35.719,Z -52.734,A 90.000,B 90.000,C 0.000} C_DIS
LIN {X -13.753,Y 35.719,Z -52.676,A 90.000,B 90.000,C 0.000} C_DIS
LIN {X -14.807,Y 35.719,Z -52.682,A 90.000,B 90.000,C 0.000} C_DIS
LIN {X -15.859,Y 35.719,Z -52.752,A 90.000,B 90.000,C 0.000} C_DIS
LIN {X -16.905,Y 35.719,Z -52.886,A 90.000,B 90.000,C 0.000} C_DIS
LIN {X -17.940,Y 35.719,Z -53.083,A 90.000,B 90.000,C 0.000} C_DIS
LIN {X -18.962,Y 35.719,Z -53.342,A 90.000,B 90.000,C 0.000} C_DIS
LIN {X -19.966,Y 35.719,Z -53.662,A 90.000,B 90.000,C 0.000} C_DIS
LIN {X -20.949,Y 35.719,Z -54.043,A 90.000,B 90.000,C 0.000} C_DIS
LIN {X -21.907,Y 35.719,Z -54.482,A 90.000,B 90.000,C 0.000} C_DIS
LIN {X -22.544,Y 35.719,Z -54.774,A 90.000,B 90.000,C 0.000} C_DIS
LIN {X -23.159,Y 35.719,Z -55.111,A 90.000,B 90.000,C 0.000} C_DIS
LIN {X -23.748,Y 35.719,Z -55.491,A 90.000,B 90.000,C 0.000} C_DIS
LIN {X -24.308,Y 35.719,Z -55.913,A 90.000,B 90.000,C 0.000} C_DIS
LIN {X -24.836,Y 35.719,Z -56.375,A 90.000,B 90.000,C 0.000} C_DIS
LIN {X -25.329,Y 35.719,Z -56.873,A 90.000,B 90.000,C 0.000} C_DIS
LIN {X -26.848,Y 35.719,Z -56.446,A 90.000,B 90.000,C 0.000} C_DIS
LIN {X -28.383,Y 35.719,Z -56.082,A 90.000,B 90.000,C 0.000} C_DIS
LIN {X -29.931,Y 35.719,Z -55.781,A 90.000,B 90.000,C 0.000} C_DIS
LIN {X -31.491,Y 35.719,Z -55.543,A 90.000,B 90.000,C 0.000} C_DIS
LIN {X -33.059,Y 35.719,Z -55.368,A 90.000,B 90.000,C 0.000} C_DIS
LIN {X -34.632,Y 35.719,Z -55.258,A 90.000,B 90.000,C 0.000} C_DIS
LIN {X -36.209,Y 35.719,Z -55.213,A 90.000,B 90.000,C 0.000} C_DIS
LIN {X -37.787,Y 35.719,Z -55.231,A 90.000,B 90.000,C 0.000} C_DIS
LIN {X -39.362,Y 35.719,Z -55.315,A 90.000,B 90.000,C 0.000} C_DIS
LIN {X -40.622,Y 35.719,Z -55.395,A 90.000,B 90.000,C 0.000} C_DIS
LIN {X -41.878,Y 35.719,Z -55.532,A 90.000,B 90.000,C 0.000} C_DIS
LIN {X -43.126,Y 35.719,Z -55.725,A 90.000,B 90.000,C 0.000} C_DIS
LIN {X -44.364,Y 35.719,Z -55.974,A 90.000,B 90.000,C 0.000} C_DIS
LIN {X -45.590,Y 35.719,Z -56.278,A 90.000,B 90.000,C 0.000} C_DIS
LIN {X -46.801,Y 35.719,Z -56.637,A 90.000,B 90.000,C 0.000} C_DIS
LIN {X -47.994,Y 35.719,Z -57.049,A 90.000,B 90.000,C 0.000} C_DIS
LIN {X -49.168,Y 35.719,Z -57.515,A 90.000,B 90.000,C 0.000} C_DIS
LIN {X -50.179,Y 35.719,Z -57.919,A 90.000,B 90.000,C 0.000} C_DIS
LIN {X -51.162,Y 35.719,Z -58.390,A 90.000,B 90.000,C 0.000} C_DIS
LIN {X -52.111,Y 35.719,Z -58.923,A 90.000,B 90.000,C 0.000} C_DIS
LIN {X -53.024,Y 35.719,Z -59.519,A 90.000,B 90.000,C 0.000} C_DIS
LIN {X -53.895,Y 35.719,Z -60.173,A 90.000,B 90.000,C 0.000} C_DIS
LIN {X -54.721,Y 35.719,Z -60.883,A 90.000,B 90.000,C 0.000} C_DIS
LIN {X -55.498,Y 35.719,Z -61.645,A 90.000,B 90.000,C 0.000} C_DIS
LIN {X -56.224,Y 35.719,Z -62.458,A 90.000,B 90.000,C 0.000} C_DIS
LIN {X -56.894,Y 35.719,Z -63.316,A 90.000,B 90.000,C 0.000} C_DIS
LIN {X -57.506,Y 35.719,Z -64.217,A 90.000,B 90.000,C 0.000} C_DIS
LIN {X -58.058,Y 35.719,Z -65.156,A 90.000,B 90.000,C 0.000} C_DIS
LIN {X -58.547,Y 35.719,Z -66.130,A 90.000,B 90.000,C 0.000} C_DIS
LIN {X -58.970,Y 35.719,Z -67.133,A 90.000,B 90.000,C 0.000} C_DIS
LIN {X -59.328,Y 35.719,Z -68.162,A 90.000,B 90.000,C 0.000} C_DIS
LIN {X -59.691,Y 35.719,Z -69.643,A 90.000,B 90.000,C 0.000} C_DIS
LIN {X -59.990,Y 35.719,Z -71.138,A 90.000,B 90.000,C 0.000} C_DIS
LIN {X -60.224,Y 35.719,Z -72.644,A 90.000,B 90.000,C 0.000} C_DIS
LIN {X -60.392,Y 35.719,Z -74.159,A 90.000,B 90.000,C 0.000} C_DIS
LIN {X -60.495,Y 35.719,Z -75.680,A 90.000,B 90.000,C 0.000} C_DIS
LIN {X -60.532,Y 35.719,Z -77.204,A 90.000,B 90.000,C 0.000} C_DIS
LIN {X -60.503,Y 35.719,Z -78.729,A 90.000,B 90.000,C 0.000} C_DIS
LIN {X -60.409,Y 35.719,Z -80.250,A 90.000,B 90.000,C 0.000} C_DIS
LIN {X -60.248,Y 35.719,Z -81.766,A 90.000,B 90.000,C 0.000} C_DIS
LIN {X -60.022,Y 35.719,Z -83.274,A 90.000,B 90.000,C 0.000} C_DIS
LIN {X -59.714,Y 35.719,Z -85.040,A 90.000,B 90.000,C 0.000} C_DIS
LIN {X -59.339,Y 35.719,Z -86.794,A 90.000,B 90.000,C 0.000} C_DIS
LIN {X -58.899,Y 35.719,Z -88.532,A 90.000,B 90.000,C 0.000} C_DIS
LIN {X -58.395,Y 35.719,Z -90.252,A 90.000,B 90.000,C 0.000} C_DIS
LIN {X -57.826,Y 35.719,Z -91.952,A 90.000,B 90.000,C 0.000} C_DIS
LIN {X -57.194,Y 35.719,Z -93.630,A 90.000,B 90.000,C 0.000} C_DIS
LIN {X -56.500,Y 35.719,Z -95.283,A 90.000,B 90.000,C 0.000} C_DIS
LIN {X -55.744,Y 35.719,Z -96.909,A 90.000,B 90.000,C 0.000} C_DIS
LIN {X -54.773,Y 35.719,Z -98.724,A 90.000,B 90.000,C 0.000} C_DIS
LIN {X -53.746,Y 35.719,Z -100.509,A 90.000,B 90.000,C 0.000} C_DIS
LIN {X -52.664,Y 35.719,Z -102.260,A 90.000,B 90.000,C 0.000} C_DIS
LIN {X -51.528,Y 35.719,Z -103.977,A 90.000,B 90.000,C 0.000} C_DIS
LIN {X -50.340,Y 35.719,Z -105.658,A 90.000,B 90.000,C 0.000} C_DIS
LIN {X -49.599,Y 35.719,Z -106.576,A 90.000,B 90.000,C 0.000} C_DIS
LIN {X -48.884,Y 35.719,Z -107.515,A 90.000,B 90.000,C 0.000} C_DIS
LIN {X -48.194,Y 35.719,Z -108.472,A 90.000,B 90.000,C 0.000} C_DIS
LIN {X -47.530,Y 35.719,Z -109.447,A 90.000,B 90.000,C 0.000} C_DIS
LIN {X -47.506,Y 35.719,Z -111.300,A 90.000,B 90.000,C 0.000} C_DIS
LIN {X -47.411,Y 35.719,Z -113.151,A 90.000,B 90.000,C 0.000} C_DIS
LIN {X -47.245,Y 35.719,Z -114.997,A 90.000,B 90.000,C 0.000} C_DIS
LIN {X -47.008,Y 35.719,Z -116.836,A 90.000,B 90.000,C 0.000} C_DIS
LIN {X -46.702,Y 35.719,Z -118.664,A 90.000,B 90.000,C 0.000} C_DIS
LIN {X -46.325,Y 35.719,Z -120.479,A 90.000,B 90.000,C 0.000} C_DIS
LIN {X -45.880,Y 35.719,Z -122.278,A 90.000,B 90.000,C 0.000} C_DIS
LIN {X -45.365,Y 35.719,Z -124.059,A 90.000,B 90.000,C 0.000} C_DIS
LIN {X -44.783,Y 35.719,Z -125.818,A 90.000,B 90.000,C 0.000} C_DIS
LIN {X -44.135,Y 35.719,Z -127.555,A 90.000,B 90.000,C 0.000} C_DIS
LIN {X -43.420,Y 35.719,Z -129.265,A 90.000,B 90.000,C 0.000} C_DIS
LIN {X -42.640,Y 35.719,Z -130.946,A 90.000,B 90.000,C 0.000} C_DIS
LIN {X -41.796,Y 35.719,Z -132.596,A 90.000,B 90.000,C 0.000} C_DIS
LIN {X -40.890,Y 35.719,Z -134.213,A 90.000,B 90.000,C 0.000} C_DIS
LIN {X -39.922,Y 35.719,Z -135.794,A 90.000,B 90.000,C 0.000} C_DIS
LIN {X -38.895,Y 35.719,Z -137.337,A 90.000,B 90.000,C 0.000} C_DIS
LIN {X -38.002,Y 35.719,Z -138.600,A 90.000,B 90.000,C 0.000} C_DIS
LIN {X -37.065,Y 35.719,Z -139.829,A 90.000,B 90.000,C 0.000} C_DIS
LIN {X -36.083,Y 35.719,Z -141.024,A 90.000,B 90.000,C 0.000} C_DIS
LIN {X -35.058,Y 35.719,Z -142.182,A 90.000,B 90.000,C 0.000} C_DIS
LIN {X -33.993,Y 35.719,Z -143.303,A 90.000,B 90.000,C 0.000} C_DIS
LIN {X -32.887,Y 35.719,Z -144.384,A 90.000,B 90.000,C 0.000} C_DIS
LIN {X -31.832,Y 35.719,Z -145.477,A 90.000,B 90.000,C 0.000} C_DIS
LIN {X -30.739,Y 35.719,Z -146.532,A 90.000,B 90.000,C 0.000} C_DIS
LIN {X -29.610,Y 35.719,Z -147.550,A 90.000,B 90.000,C 0.000} C_DIS
LIN {X -28.447,Y 35.719,Z -148.527,A 90.000,B 90.000,C 0.000} C_DIS
LIN {X -27.250,Y 35.719,Z -149.463,A 90.000,B 90.000,C 0.000} C_DIS
LIN {X -26.022,Y 35.719,Z -150.357,A 90.000,B 90.000,C 0.000} C_DIS
LIN {X -24.297,Y 35.719,Z -151.682,A 90.000,B 90.000,C 0.000} C_DIS
LIN {X -22.530,Y 35.719,Z -152.951,A 90.000,B 90.000,C 0.000} C_DIS
LIN {X -20.722,Y 35.719,Z -154.160,A 90.000,B 90.000,C 0.000} C_DIS
LIN {X -18.875,Y 35.719,Z -155.310,A 90.000,B 90.000,C 0.000} C_DIS
LIN {X -16.992,Y 35.719,Z -156.399,A 90.000,B 90.000,C 0.000} C_DIS
LIN {X -15.074,Y 35.719,Z -157.425,A 90.000,B 90.000,C 0.000} C_DIS
LIN {X -13.123,Y 35.719,Z -158.388,A 90.000,B 90.000,C 0.000} C_DIS
LIN {X -11.142,Y 35.719,Z -159.286,A 90.000,B 90.000,C 0.000} C_DIS
LIN {X -9.133,Y 35.719,Z -160.120,A 90.000,B 90.000,C 0.000} C_DIS
LIN {X -7.097,Y 35.719,Z -160.886,A 90.000,B 90.000,C 0.000} C_DIS
LIN {X -5.037,Y 35.719,Z -161.586,A 90.000,B 90.000,C 0.000} C_DIS
LIN {X -2.956,Y 35.719,Z -162.219,A 90.000,B 90.000,C 0.000} C_DIS
LIN {X -2.087,Y 35.719,Z -162.590,A 90.000,B 90.000,C 0.000} C_DIS
LIN {X -1.204,Y 35.719,Z -162.925,A 90.000,B 90.000,C 0.000} C_DIS
LIN {X -0.307,Y 35.719,Z -163.222,A 90.000,B 90.000,C 0.000} C_DIS
LIN {X 0.601,Y 35.719,Z -163.480,A 90.000,B 90.000,C 0.000} C_DIS
LIN {X 1.520,Y 35.719,Z -163.700,A 90.000,B 90.000,C 0.000} C_DIS
LIN {X 1.881,Y 35.719,Z -163.789,A 90.000,B 90.000,C 0.000} C_DIS
LIN {X 2.227,Y 35.719,Z -163.923,A 90.000,B 90.000,C 0.000} C_DIS
LIN {X 2.553,Y 35.719,Z -164.101,A 90.000,B 90.000,C 0.000} C_DIS
LIN {X 2.854,Y 35.719,Z -164.320,A 90.000,B 90.000,C 0.000} C_DIS
LIN {X 3.123,Y 35.719,Z -164.576,A 90.000,B 90.000,C 0.000} C_DIS
LIN {X 3.357,Y 35.719,Z -164.865,A 90.000,B 90.000,C 0.000} C_DIS
LIN {X 3.431,Y 35.719,Z -165.010,A 90.000,B 90.000,C 0.000} C_DIS
LIN {X 3.537,Y 35.719,Z -165.365,A 90.000,B 90.000,C 0.000} C_DIS
LIN {X 3.602,Y 35.719,Z -165.731,A 90.000,B 90.000,C 0.000} C_DIS
LIN {X 3.624,Y 35.719,Z -166.101,A 90.000,B 90.000,C 0.000} C_DIS
LIN {X 3.282,Y 35.719,Z -166.833,A 90.000,B 90.000,C 0.000} C_DIS
LIN {X 2.893,Y 35.719,Z -167.541,A 90.000,B 90.000,C 0.000} C_DIS
LIN {X 2.460,Y 35.719,Z -168.223,A 90.000,B 90.000,C 0.000} C_DIS
LIN {X 1.985,Y 35.719,Z -168.876,A 90.000,B 90.000,C 0.000} C_DIS
LIN {X 1.468,Y 35.719,Z -169.497,A 90.000,B 90.000,C 0.000} C_DIS
LIN {X 0.913,Y 35.719,Z -170.084,A 90.000,B 90.000,C 0.000} C_DIS
LIN {X -1.717,Y 35.719,Z -172.736,A 90.000,B 90.000,C 0.000} C_DIS
LIN {X -4.393,Y 35.719,Z -175.342,A 90.000,B 90.000,C 0.000} C_DIS
LIN {X -7.114,Y 35.719,Z -177.902,A 90.000,B 90.000,C 0.000} C_DIS
LIN {X -9.878,Y 35.719,Z -180.414,A 90.000,B 90.000,C 0.000} C_DIS
LIN {X -12.686,Y 35.719,Z -182.877,A 90.000,B 90.000,C 0.000} C_DIS
LIN {X -15.536,Y 35.719,Z -185.292,A 90.000,B 90.000,C 0.000} C_DIS
LIN {X -18.427,Y 35.719,Z -187.657,A 90.000,B 90.000,C 0.000} C_DIS
LIN {X -21.359,Y 35.719,Z -189.971,A 90.000,B 90.000,C 0.000} C_DIS
LIN {X -24.330,Y 35.719,Z -192.235,A 90.000,B 90.000,C 0.000} C_DIS
LIN {X -27.026,Y 35.719,Z -194.106,A 90.000,B 90.000,C 0.000} C_DIS
LIN {X -29.760,Y 35.719,Z -195.921,A 90.000,B 90.000,C 0.000} C_DIS
LIN {X -32.530,Y 35.719,Z -197.680,A 90.000,B 90.000,C 0.000} C_DIS
LIN {X -35.335,Y 35.719,Z -199.382,A 90.000,B 90.000,C 0.000} C_DIS
LIN {X -38.175,Y 35.719,Z -201.026,A 90.000,B 90.000,C 0.000} C_DIS
LIN {X -41.048,Y 35.719,Z -202.612,A 90.000,B 90.000,C 0.000} C_DIS
LIN {X -43.953,Y 35.719,Z -204.139,A 90.000,B 90.000,C 0.000} C_DIS
LIN {X -46.888,Y 35.719,Z -205.606,A 90.000,B 90.000,C 0.000} C_DIS
LIN {X -51.874,Y 35.719,Z -208.102,A 90.000,B 90.000,C 0.000} C_DIS
LIN {X -55.959,Y 35.719,Z -210.035,A 90.000,B 90.000,C 0.000} C_DIS
LIN {X -60.016,Y 35.719,Z -212.029,A 90.000,B 90.000,C 0.000} C_DIS
LIN {X -64.042,Y 35.719,Z -214.081,A 90.000,B 90.000,C 0.000} C_DIS
LIN {X -68.038,Y 35.719,Z -216.193,A 90.000,B 90.000,C 0.000} C_DIS
LIN {X -72.003,Y 35.719,Z -218.364,A 90.000,B 90.000,C 0.000} C_DIS
LIN {X -75.934,Y 35.719,Z -220.593,A 90.000,B 90.000,C 0.000} C_DIS
LIN {X -79.833,Y 35.719,Z -222.880,A 90.000,B 90.000,C 0.000} C_DIS
LIN {X -83.697,Y 35.719,Z -225.224,A 90.000,B 90.000,C 0.000} C_DIS
LIN {X -87.527,Y 35.719,Z -227.624,A 90.000,B 90.000,C 0.000} C_DIS
LIN {X -91.320,Y 35.719,Z -230.081,A 90.000,B 90.000,C 0.000} C_DIS
LIN {X -95.077,Y 35.719,Z -232.594,A 90.000,B 90.000,C 0.000} C_DIS
LIN {X -98.797,Y 35.719,Z -235.162,A 90.000,B 90.000,C 0.000} C_DIS
LIN {X -102.478,Y 35.719,Z -237.784,A 90.000,B 90.000,C 0.000} C_DIS
LIN {X -104.422,Y 35.719,Z -239.171,A 90.000,B 90.000,C 0.000} C_DIS
LIN {X -106.337,Y 35.719,Z -240.596,A 90.000,B 90.000,C 0.000} C_DIS
LIN {X -108.224,Y 35.719,Z -242.060,A 90.000,B 90.000,C 0.000} C_DIS
LIN {X -110.081,Y 35.719,Z -243.561,A 90.000,B 90.000,C 0.000} C_DIS
LIN {X -145.015,Y 35.719,Z -243.561,A 90.000,B 90.000,C 0.000} C_DIS
LIN {X -145.015,Y 35.719,Z 0.000,A 90.000,B 90.000,C 0.000} C_DIS
LIN {X 145.015,Y 35.719,Z 0.000,A 90.000,B 90.000,C 0.000} C_DIS
LIN {X 145.015,Y 35.719,Z -243.561,A 90.000,B 90.000,C 0.000} C_DIS
LIN {X 69.937,Y 35.719,Z -243.561,A 90.000,B 90.000,C 0.000} C_DIS
LIN {X 71.997,Y 35.719,Z -238.419,A 90.000,B 90.000,C 0.000} C_DIS
LIN {X 72.589,Y 35.719,Z -237.047,A 90.000,B 90.000,C 0.000} C_DIS
LIN {X 73.159,Y 35.719,Z -235.665,A 90.000,B 90.000,C 0.000} C_DIS
LIN {X 73.708,Y 35.719,Z -234.275,A 90.000,B 90.000,C 0.000} C_DIS
LIN {X 75.762,Y 35.719,Z -229.564,A 90.000,B 90.000,C 0.000} C_DIS
LIN {X 77.761,Y 35.719,Z -224.829,A 90.000,B 90.000,C 0.000} C_DIS
LIN {X 79.705,Y 35.719,Z -220.071,A 90.000,B 90.000,C 0.000} C_DIS
LIN {X 81.593,Y 35.719,Z -215.291,A 90.000,B 90.000,C 0.000} C_DIS
LIN {X 83.425,Y 35.719,Z -210.489,A 90.000,B 90.000,C 0.000} C_DIS
LIN {X 85.202,Y 35.719,Z -205.667,A 90.000,B 90.000,C 0.000} C_DIS
LIN {X 86.922,Y 35.719,Z -200.824,A 90.000,B 90.000,C 0.000} C_DIS
LIN {X 88.585,Y 35.719,Z -195.961,A 90.000,B 90.000,C 0.000} C_DIS
LIN {X 90.192,Y 35.719,Z -191.079,A 90.000,B 90.000,C 0.000} C_DIS
LIN {X 91.743,Y 35.719,Z -186.179,A 90.000,B 90.000,C 0.000} C_DIS
LIN {X 94.599,Y 35.719,Z -177.190,A 90.000,B 90.000,C 0.000} C_DIS
LIN {X 95.482,Y 35.719,Z -174.477,A 90.000,B 90.000,C 0.000} C_DIS
LIN {X 96.318,Y 35.719,Z -171.750,A 90.000,B 90.000,C 0.000} C_DIS
LIN {X 97.106,Y 35.719,Z -169.008,A 90.000,B 90.000,C 0.000} C_DIS
LIN {X 97.846,Y 35.719,Z -166.253,A 90.000,B 90.000,C 0.000} C_DIS
LIN {X 98.538,Y 35.719,Z -163.485,A 90.000,B 90.000,C 0.000} C_DIS
LIN {X 99.181,Y 35.719,Z -160.706,A 90.000,B 90.000,C 0.000} C_DIS
LIN {X 99.776,Y 35.719,Z -157.916,A 90.000,B 90.000,C 0.000} C_DIS
LIN {X 100.393,Y 35.719,Z -154.125,A 90.000,B 90.000,C 0.000} C_DIS
LIN {X 100.951,Y 35.719,Z -150.324,A 90.000,B 90.000,C 0.000} C_DIS
LIN {X 101.449,Y 35.719,Z -146.515,A 90.000,B 90.000,C 0.000} C_DIS
LIN {X 101.888,Y 35.719,Z -142.699,A 90.000,B 90.000,C 0.000} C_DIS
LIN {X 102.266,Y 35.719,Z -138.876,A 90.000,B 90.000,C 0.000} C_DIS
LIN {X 102.584,Y 35.719,Z -135.048,A 90.000,B 90.000,C 0.000} C_DIS
LIN {X 102.843,Y 35.719,Z -132.585,A 90.000,B 90.000,C 0.000} C_DIS
LIN {X 103.043,Y 35.719,Z -130.117,A 90.000,B 90.000,C 0.000} C_DIS
LIN {X 103.183,Y 35.719,Z -127.644,A 90.000,B 90.000,C 0.000} C_DIS
LIN {X 103.264,Y 35.719,Z -125.169,A 90.000,B 90.000,C 0.000} C_DIS
LIN {X 103.285,Y 35.719,Z -122.692,A 90.000,B 90.000,C 0.000} C_DIS
LIN {X 103.247,Y 35.719,Z -120.216,A 90.000,B 90.000,C 0.000} C_DIS
LIN {X 103.185,Y 35.719,Z -117.560,A 90.000,B 90.000,C 0.000} C_DIS
LIN {X 103.141,Y 35.719,Z -114.904,A 90.000,B 90.000,C 0.000} C_DIS
LIN {X 103.193,Y 35.719,Z -113.235,A 90.000,B 90.000,C 0.000} C_DIS
LIN {X 103.191,Y 35.719,Z -111.565,A 90.000,B 90.000,C 0.000} C_DIS
LIN {X 103.135,Y 35.719,Z -109.895,A 90.000,B 90.000,C 0.000} C_DIS
LIN {X 103.024,Y 35.719,Z -108.229,A 90.000,B 90.000,C 0.000} C_DIS
LIN {X 102.859,Y 35.719,Z -106.567,A 90.000,B 90.000,C 0.000} C_DIS
LIN {X 102.641,Y 35.719,Z -104.911,A 90.000,B 90.000,C 0.000} C_DIS
LIN {X 102.805,Y 35.719,Z -104.116,A 90.000,B 90.000,C 0.000} C_DIS
LIN {X 102.993,Y 35.719,Z -103.326,A 90.000,B 90.000,C 0.000} C_DIS
LIN {X 103.203,Y 35.719,Z -102.542,A 90.000,B 90.000,C 0.000} C_DIS
LIN {X 103.639,Y 35.719,Z -101.218,A 90.000,B 90.000,C 0.000} C_DIS
LIN {X 104.035,Y 35.719,Z -99.881,A 90.000,B 90.000,C 0.000} C_DIS
LIN {X 104.392,Y 35.719,Z -98.534,A 90.000,B 90.000,C 0.000} C_DIS
LIN {X 104.709,Y 35.719,Z -97.176,A 90.000,B 90.000,C 0.000} C_DIS
LIN {X 104.998,Y 35.719,Z -94.571,A 90.000,B 90.000,C 0.000} C_DIS
LIN {X 105.250,Y 35.719,Z -91.963,A 90.000,B 90.000,C 0.000} C_DIS
LIN {X 105.466,Y 35.719,Z -89.351,A 90.000,B 90.000,C 0.000} C_DIS
LIN {X 106.785,Y 35.719,Z -87.443,A 90.000,B 90.000,C 0.000} C_DIS
LIN {X 108.046,Y 35.719,Z -85.496,A 90.000,B 90.000,C 0.000} C_DIS
LIN {X 109.247,Y 35.719,Z -83.512,A 90.000,B 90.000,C 0.000} C_DIS
LIN {X 110.387,Y 35.719,Z -81.493,A 90.000,B 90.000,C 0.000} C_DIS
LIN {X 111.466,Y 35.719,Z -79.440,A 90.000,B 90.000,C 0.000} C_DIS
LIN {X 112.482,Y 35.719,Z -77.355,A 90.000,B 90.000,C 0.000} C_DIS
LIN {X 113.435,Y 35.719,Z -75.240,A 90.000,B 90.000,C 0.000} C_DIS
LIN {X 114.323,Y 35.719,Z -73.098,A 90.000,B 90.000,C 0.000} C_DIS
LIN {X 115.146,Y 35.719,Z -70.929,A 90.000,B 90.000,C 0.000} C_DIS
LIN {X 115.903,Y 35.719,Z -68.737,A 90.000,B 90.000,C 0.000} C_DIS
LIN {X 116.594,Y 35.719,Z -66.523,A 90.000,B 90.000,C 0.000} C_DIS
LIN {X 117.007,Y 35.719,Z -64.737,A 90.000,B 90.000,C 0.000} C_DIS
LIN {X 117.487,Y 35.719,Z -62.967,A 90.000,B 90.000,C 0.000} C_DIS
LIN {X 118.033,Y 35.719,Z -61.216,A 90.000,B 90.000,C 0.000} C_DIS
LIN {X 118.644,Y 35.719,Z -59.488,A 90.000,B 90.000,C 0.000} C_DIS
LIN {X 119.320,Y 35.719,Z -57.783,A 90.000,B 90.000,C 0.000} C_DIS
LIN {X 120.059,Y 35.719,Z -56.105,A 90.000,B 90.000,C 0.000} C_DIS
LIN {X 120.861,Y 35.719,Z -54.456,A 90.000,B 90.000,C 0.000} C_DIS
LIN {X 121.447,Y 35.719,Z -53.407,A 90.000,B 90.000,C 0.000} C_DIS
LIN {X 121.988,Y 35.719,Z -52.335,A 90.000,B 90.000,C 0.000} C_DIS
LIN {X 122.484,Y 35.719,Z -51.242,A 90.000,B 90.000,C 0.000} C_DIS
LIN {X 122.934,Y 35.719,Z -50.128,A 90.000,B 90.000,C 0.000} C_DIS
LIN {X 123.338,Y 35.719,Z -48.997,A 90.000,B 90.000,C 0.000} C_DIS
LIN {X 123.694,Y 35.719,Z -47.850,A 90.000,B 90.000,C 0.000} C_DIS
LIN {X 123.995,Y 35.719,Z -46.793,A 90.000,B 90.000,C 0.000} C_DIS
LIN {X 124.225,Y 35.719,Z -45.719,A 90.000,B 90.000,C 0.000} C_DIS
LIN {X 124.383,Y 35.719,Z -44.632,A 90.000,B 90.000,C 0.000} C_DIS
LIN {X 124.469,Y 35.719,Z -43.537,A 90.000,B 90.000,C 0.000} C_DIS
LIN {X 124.482,Y 35.719,Z -42.439,A 90.000,B 90.000,C 0.000} C_DIS
LIN {X 124.423,Y 35.719,Z -41.342,A 90.000,B 90.000,C 0.000} C_DIS
LIN {X 124.290,Y 35.719,Z -40.252,A 90.000,B 90.000,C 0.000} C_DIS
LIN {X 124.086,Y 35.719,Z -39.172,A 90.000,B 90.000,C 0.000} C_DIS
LIN {X 123.811,Y 35.719,Z -38.109,A 90.000,B 90.000,C 0.000} C_DIS
LIN {X 123.466,Y 35.719,Z -37.066,A 90.000,B 90.000,C 0.000} C_DIS
LIN {X 123.414,Y 35.719,Z -36.923,A 90.000,B 90.000,C 0.000} C_DIS
LIN {X 123.032,Y 35.719,Z -36.046,A 90.000,B 90.000,C 0.000} C_DIS
LIN {X 122.588,Y 35.719,Z -35.200,A 90.000,B 90.000,C 0.000} C_DIS
LIN {X 122.083,Y 35.719,Z -34.387,A 90.000,B 90.000,C 0.000} C_DIS
LIN {X 121.522,Y 35.719,Z -33.614,A 90.000,B 90.000,C 0.000} C_DIS
LIN {X 120.906,Y 35.719,Z -32.882,A 90.000,B 90.000,C 0.000} C_DIS
LIN {X 120.239,Y 35.719,Z -32.197,A 90.000,B 90.000,C 0.000} C_DIS
LIN {X 119.524,Y 35.719,Z -31.562,A 90.000,B 90.000,C 0.000} C_DIS
LIN {X 118.765,Y 35.719,Z -30.980,A 90.000,B 90.000,C 0.000} C_DIS
LIN {X 117.966,Y 35.719,Z -30.455,A 90.000,B 90.000,C 0.000} C_DIS
LIN {X 117.834,Y 35.719,Z -30.373,A 90.000,B 90.000,C 0.000} C_DIS
LIN {X 117.055,Y 35.719,Z -29.942,A 90.000,B 90.000,C 0.000} C_DIS
LIN {X 116.250,Y 35.719,Z -29.561,A 90.000,B 90.000,C 0.000} C_DIS
LIN {X 115.424,Y 35.719,Z -29.230,A 90.000,B 90.000,C 0.000} C_DIS
LIN {X 114.578,Y 35.719,Z -28.952,A 90.000,B 90.000,C 0.000} C_DIS
LIN {X 114.396,Y 35.719,Z -28.894,A 90.000,B 90.000,C 0.000} C_DIS
LIN {X 113.513,Y 35.719,Z -28.671,A 90.000,B 90.000,C 0.000} C_DIS
LIN {X 112.617,Y 35.719,Z -28.507,A 90.000,B 90.000,C 0.000} C_DIS
LIN {X 111.712,Y 35.719,Z -28.400,A 90.000,B 90.000,C 0.000} C_DIS
LIN {X 110.802,Y 35.719,Z -28.353,A 90.000,B 90.000,C 0.000} C_DIS
LIN {X 109.891,Y 35.719,Z -28.364,A 90.000,B 90.000,C 0.000} C_DIS
LIN {X 108.983,Y 35.719,Z -28.435,A 90.000,B 90.000,C 0.000} C_DIS
LIN {X 108.081,Y 35.719,Z -28.564,A 90.000,B 90.000,C 0.000} C_DIS
LIN {X 107.190,Y 35.719,Z -28.752,A 90.000,B 90.000,C 0.000} C_DIS
LIN {X 105.045,Y 35.719,Z -29.510,A 90.000,B 90.000,C 0.000} C_DIS
LIN {X 102.919,Y 35.719,Z -30.321,A 90.000,B 90.000,C 0.000} C_DIS
LIN {X 100.814,Y 35.719,Z -31.185,A 90.000,B 90.000,C 0.000} C_DIS
LIN {X 98.731,Y 35.719,Z -32.101,A 90.000,B 90.000,C 0.000} C_DIS
LIN {X 96.671,Y 35.719,Z -33.068,A 90.000,B 90.000,C 0.000} C_DIS
LIN {X 95.620,Y 35.719,Z -33.535,A 90.000,B 90.000,C 0.000} C_DIS
LIN {X 94.599,Y 35.719,Z -34.066,A 90.000,B 90.000,C 0.000} C_DIS
LIN {X 93.612,Y 35.719,Z -34.657,A 90.000,B 90.000,C 0.000} C_DIS
LIN {X 92.663,Y 35.719,Z -35.307,A 90.000,B 90.000,C 0.000} C_DIS
LIN {X 91.755,Y 35.719,Z -36.013,A 90.000,B 90.000,C 0.000} C_DIS
LIN {X 90.891,Y 35.719,Z -36.773,A 90.000,B 90.000,C 0.000} C_DIS
LIN {X 90.075,Y 35.719,Z -37.583,A 90.000,B 90.000,C 0.000} C_DIS
LIN {X 89.309,Y 35.719,Z -38.442,A 90.000,B 90.000,C 0.000} C_DIS
LIN {X 88.752,Y 35.719,Z -39.121,A 90.000,B 90.000,C 0.000} C_DIS
LIN {X 88.241,Y 35.719,Z -39.834,A 90.000,B 90.000,C 0.000} C_DIS
LIN {X 87.778,Y 35.719,Z -40.579,A 90.000,B 90.000,C 0.000} C_DIS
LIN {X 87.364,Y 35.719,Z -41.354,A 90.000,B 90.000,C 0.000} C_DIS
LIN {X 87.002,Y 35.719,Z -42.153,A 90.000,B 90.000,C 0.000} C_DIS
LIN {X 86.694,Y 35.719,Z -42.975,A 90.000,B 90.000,C 0.000} C_DIS
LIN {X 86.439,Y 35.719,Z -43.815,A 90.000,B 90.000,C 0.000} C_DIS
LIN {X 86.240,Y 35.719,Z -44.670,A 90.000,B 90.000,C 0.000} C_DIS
LIN {X 86.099,Y 35.719,Z -45.536,A 90.000,B 90.000,C 0.000} C_DIS
LIN {X 86.002,Y 35.719,Z -46.184,A 90.000,B 90.000,C 0.000} C_DIS
LIN {X 85.966,Y 35.719,Z -46.838,A 90.000,B 90.000,C 0.000} C_DIS
LIN {X 85.993,Y 35.719,Z -47.493,A 90.000,B 90.000,C 0.000} C_DIS
LIN {X 86.081,Y 35.719,Z -48.142,A 90.000,B 90.000,C 0.000} C_DIS
LIN {X 84.784,Y 35.719,Z -49.229,A 90.000,B 90.000,C 0.000} C_DIS
LIN {X 83.530,Y 35.719,Z -50.366,A 90.000,B 90.000,C 0.000} C_DIS
LIN {X 82.321,Y 35.719,Z -51.550,A 90.000,B 90.000,C 0.000} C_DIS
LIN {X 81.159,Y 35.719,Z -52.781,A 90.000,B 90.000,C 0.000} C_DIS
LIN {X 80.046,Y 35.719,Z -54.056,A 90.000,B 90.000,C 0.000} C_DIS
LIN {X 78.984,Y 35.719,Z -55.373,A 90.000,B 90.000,C 0.000} C_DIS
LIN {X 77.973,Y 35.719,Z -56.731,A 90.000,B 90.000,C 0.000} C_DIS
LIN {X 77.016,Y 35.719,Z -58.127,A 90.000,B 90.000,C 0.000} C_DIS
LIN {X 76.062,Y 35.719,Z -56.940,A 90.000,B 90.000,C 0.000} C_DIS
LIN {X 75.965,Y 35.719,Z -56.835,A 90.000,B 90.000,C 0.000} C_DIS
LIN {X 74.282,Y 35.719,Z -55.182,A 90.000,B 90.000,C 0.000} C_DIS
LIN {X 72.565,Y 35.719,Z -53.562,A 90.000,B 90.000,C 0.000} C_DIS
LIN {X 70.817,Y 35.719,Z -51.978,A 90.000,B 90.000,C 0.000} C_DIS
LIN {X 69.036,Y 35.719,Z -50.430,A 90.000,B 90.000,C 0.000} C_DIS
LIN {X 67.272,Y 35.719,Z -48.756,A 90.000,B 90.000,C 0.000} C_DIS
LIN {X 65.483,Y 35.719,Z -47.108,A 90.000,B 90.000,C 0.000} C_DIS
LIN {X 63.669,Y 35.719,Z -45.488,A 90.000,B 90.000,C 0.000} C_DIS
LIN {X 61.830,Y 35.719,Z -43.896,A 90.000,B 90.000,C 0.000} C_DIS
LIN {X 60.860,Y 35.719,Z -43.106,A 90.000,B 90.000,C 0.000} C_DIS
LIN {X 59.852,Y 35.719,Z -42.367,A 90.000,B 90.000,C 0.000} C_DIS
LIN {X 58.807,Y 35.719,Z -41.679,A 90.000,B 90.000,C 0.000} C_DIS
LIN {X 57.729,Y 35.719,Z -41.045,A 90.000,B 90.000,C 0.000} C_DIS
LIN {X 56.621,Y 35.719,Z -40.467,A 90.000,B 90.000,C 0.000} C_DIS
LIN {X 55.484,Y 35.719,Z -39.945,A 90.000,B 90.000,C 0.000} C_DIS
LIN {X 54.322,Y 35.719,Z -39.482,A 90.000,B 90.000,C 0.000} C_DIS
LIN {X 53.139,Y 35.719,Z -39.078,A 90.000,B 90.000,C 0.000} C_DIS
LIN {X 51.936,Y 35.719,Z -38.735,A 90.000,B 90.000,C 0.000} C_DIS
LIN {X 50.718,Y 35.719,Z -38.453,A 90.000,B 90.000,C 0.000} C_DIS
LIN {X 50.555,Y 35.719,Z -38.428,A 90.000,B 90.000,C 0.000} C_DIS
LIN {X 49.479,Y 35.719,Z -38.308,A 90.000,B 90.000,C 0.000} C_DIS
LIN {X 48.399,Y 35.719,Z -38.249,A 90.000,B 90.000,C 0.000} C_DIS
LIN {X 47.317,Y 35.719,Z -38.250,A 90.000,B 90.000,C 0.000} C_DIS
LIN {X 46.236,Y 35.719,Z -38.311,A 90.000,B 90.000,C 0.000} C_DIS
LIN {X 45.161,Y 35.719,Z -38.432,A 90.000,B 90.000,C 0.000} C_DIS
LIN {X 44.094,Y 35.719,Z -38.613,A 90.000,B 90.000,C 0.000} C_DIS
LIN {X 43.039,Y 35.719,Z -38.853,A 90.000,B 90.000,C 0.000} C_DIS
LIN {X 42.495,Y 35.719,Z -39.036,A 90.000,B 90.000,C 0.000} C_DIS
LIN {X 41.937,Y 35.719,Z -39.168,A 90.000,B 90.000,C 0.000} C_DIS
LIN {X 41.369,Y 35.719,Z -39.248,A 90.000,B 90.000,C 0.000} C_DIS
LIN {X 40.796,Y 35.719,Z -39.275,A 90.000,B 90.000,C 0.000} C_DIS
LIN {X 40.224,Y 35.719,Z -39.249,A 90.000,B 90.000,C 0.000} C_DIS
LIN {X 39.655,Y 35.719,Z -39.171,A 90.000,B 90.000,C 0.000} C_DIS
LIN {X 39.097,Y 35.719,Z -39.040,A 90.000,B 90.000,C 0.000} C_DIS
LIN {X 38.112,Y 35.719,Z -38.886,A 90.000,B 90.000,C 0.000} C_DIS
LIN {X 37.119,Y 35.719,Z -38.795,A 90.000,B 90.000,C 0.000} C_DIS
LIN {X 36.122,Y 35.719,Z -38.767,A 90.000,B 90.000,C 0.000} C_DIS
LIN {X 35.125,Y 35.719,Z -38.801,A 90.000,B 90.000,C 0.000} C_DIS
LIN {X 34.132,Y 35.719,Z -38.898,A 90.000,B 90.000,C 0.000} C_DIS
LIN {X 33.148,Y 35.719,Z -39.057,A 90.000,B 90.000,C 0.000} C_DIS
LIN {X 32.175,Y 35.719,Z -39.278,A 90.000,B 90.000,C 0.000} C_DIS
LIN {X 31.219,Y 35.719,Z -39.560,A 90.000,B 90.000,C 0.000} C_DIS
LIN {X 30.282,Y 35.719,Z -39.902,A 90.000,B 90.000,C 0.000} C_DIS
LIN {X 29.368,Y 35.719,Z -40.302,A 90.000,B 90.000,C 0.000} C_DIS
LIN {X 28.482,Y 35.719,Z -40.759,A 90.000,B 90.000,C 0.000} C_DIS
LIN {X 27.704,Y 35.719,Z -41.212,A 90.000,B 90.000,C 0.000} C_DIS
LIN {X 26.959,Y 35.719,Z -41.717,A 90.000,B 90.000,C 0.000} C_DIS
LIN {X 26.250,Y 35.719,Z -42.272,A 90.000,B 90.000,C 0.000} C_DIS
LIN {X 25.582,Y 35.719,Z -42.875,A 90.000,B 90.000,C 0.000} C_DIS
LIN {X 24.956,Y 35.719,Z -43.522,A 90.000,B 90.000,C 0.000} C_DIS
LIN {X 24.377,Y 35.719,Z -44.211,A 90.000,B 90.000,C 0.000} C_DIS
LIN {X 23.846,Y 35.719,Z -44.939,A 90.000,B 90.000,C 0.000} C_DIS
LIN {X 23.367,Y 35.719,Z -45.701,A 90.000,B 90.000,C 0.000} C_DIS
LIN {X 22.942,Y 35.719,Z -46.494,A 90.000,B 90.000,C 0.000} C_DIS
LIN {X 22.572,Y 35.719,Z -47.315,A 90.000,B 90.000,C 0.000} C_DIS
LIN {X 22.259,Y 35.719,Z -48.159,A 90.000,B 90.000,C 0.000} C_DIS
LIN {X 21.694,Y 35.719,Z -48.680,A 90.000,B 90.000,C 0.000} C_DIS
LIN {X 21.166,Y 35.719,Z -49.236,A 90.000,B 90.000,C 0.000} C_DIS
LIN {X 20.675,Y 35.719,Z -49.827,A 90.000,B 90.000,C 0.000} C_DIS
LIN {X 20.224,Y 35.719,Z -50.449,A 90.000,B 90.000,C 0.000} C_DIS
LIN {X 19.816,Y 35.719,Z -51.099,A 90.000,B 90.000,C 0.000} C_DIS
LIN {X 19.451,Y 35.719,Z -51.775,A 90.000,B 90.000,C 0.000} C_DIS
LIN {X 19.133,Y 35.719,Z -52.474,A 90.000,B 90.000,C 0.000} C_DIS
LIN {X 18.505,Y 35.719,Z -52.570,A 90.000,B 90.000,C 0.000} C_DIS
LIN {X 17.885,Y 35.719,Z -52.705,A 90.000,B 90.000,C 0.000} C_DIS
LIN {X 17.275,Y 35.719,Z -52.878,A 90.000,B 90.000,C 0.000} C_DIS
LIN {X 16.676,Y 35.719,Z -53.090,A 90.000,B 90.000,C 0.000} C_DIS
LIN {X 16.501,Y 35.719,Z -53.170,A 90.000,B 90.000,C 0.000} C_DIS
LIN {X 15.714,Y 35.719,Z -53.174,A 90.000,B 90.000,C 0.000} C_DIS
LIN {X 14.927,Y 35.719,Z -53.198,A 90.000,B 90.000,C 0.000} C_DIS
LIN {X 13.925,Y 35.719,Z -53.375,A 90.000,B 90.000,C 0.000} C_DIS
LIN {X 12.935,Y 35.719,Z -53.606,A 90.000,B 90.000,C 0.000} C_DIS
LIN {X 11.958,Y 35.719,Z -53.890,A 90.000,B 90.000,C 0.000} C_DIS
LIN {X 10.998,Y 35.719,Z -54.226,A 90.000,B 90.000,C 0.000} C_DIS
LIN {X 10.057,Y 35.719,Z -54.613,A 90.000,B 90.000,C 0.000} C_DIS
LIN {X 9.139,Y 35.719,Z -55.051,A 90.000,B 90.000,C 0.000} C_DIS
LIN {X 9.139,Y 48.219,Z -55.051,A 90.000,B 90.000,C 0.000} C_DIS
LIN {X 9.139,Y 60.719,Z -55.051,A 90.000,B 90.000,C 0.000} C_DIS
LIN {X -117.492,Y 60.719,Z -242.561,A 90.000,B 90.000,C 0.000} C_DIS
LIN {X -117.492,Y 53.575,Z -242.561,A 90.000,B 90.000,C 0.000} C_DIS
LIN {X -117.492,Y 41.075,Z -242.561,A 90.000,B 90.000,C 0.000} C_DIS
LIN {X -117.492,Y 28.575,Z -242.561,A 90.000,B 90.000,C 0.000} C_DIS
LIN {X -144.015,Y 28.575,Z -242.561,A 90.000,B 90.000,C 0.000} C_DIS
LIN {X -144.015,Y 28.575,Z -235.012,A 90.000,B 90.000,C 0.000} C_DIS
LIN {X -106.570,Y 28.575,Z -235.012,A 90.000,B 90.000,C 0.000} C_DIS
LIN {X -102.815,Y 28.575,Z -232.454,A 90.000,B 90.000,C 0.000} C_DIS
LIN {X -99.033,Y 28.575,Z -229.938,A 90.000,B 90.000,C 0.000} C_DIS
LIN {X -95.222,Y 28.575,Z -227.464,A 90.000,B 90.000,C 0.000} C_DIS
LIN {X -144.015,Y 28.575,Z -227.464,A 90.000,B 90.000,C 0.000} C_DIS
LIN {X -144.015,Y 28.575,Z -219.915,A 90.000,B 90.000,C 0.000} C_DIS
LIN {X -83.226,Y 28.575,Z -219.915,A 90.000,B 90.000,C 0.000} C_DIS
LIN {X -79.093,Y 28.575,Z -217.370,A 90.000,B 90.000,C 0.000} C_DIS
LIN {X -74.943,Y 28.575,Z -214.854,A 90.000,B 90.000,C 0.000} C_DIS
LIN {X -70.776,Y 28.575,Z -212.366,A 90.000,B 90.000,C 0.000} C_DIS
LIN {X -144.015,Y 28.575,Z -212.366,A 90.000,B 90.000,C 0.000} C_DIS
LIN {X -144.015,Y 28.575,Z -204.817,A 90.000,B 90.000,C 0.000} C_DIS
LIN {X -57.722,Y 28.575,Z -204.817,A 90.000,B 90.000,C 0.000} C_DIS
LIN {X -55.651,Y 28.575,Z -203.653,A 90.000,B 90.000,C 0.000} C_DIS
LIN {X -53.576,Y 28.575,Z -202.497,A 90.000,B 90.000,C 0.000} C_DIS
LIN {X -50.535,Y 28.575,Z -200.776,A 90.000,B 90.000,C 0.000} C_DIS
LIN {X -47.507,Y 28.575,Z -199.033,A 90.000,B 90.000,C 0.000} C_DIS
LIN {X -44.491,Y 28.575,Z -197.269,A 90.000,B 90.000,C 0.000} C_DIS
LIN {X -144.015,Y 28.575,Z -197.269,A 90.000,B 90.000,C 0.000} C_DIS
LIN {X -144.015,Y 28.575,Z -189.720,A 90.000,B 90.000,C 0.000} C_DIS
LIN {X -32.325,Y 28.575,Z -189.720,A 90.000,B 90.000,C 0.000} C_DIS
LIN {X -30.760,Y 28.575,Z -188.565,A 90.000,B 90.000,C 0.000} C_DIS
LIN {X -29.226,Y 28.575,Z -187.367,A 90.000,B 90.000,C 0.000} C_DIS
LIN {X -27.727,Y 28.575,Z -186.128,A 90.000,B 90.000,C 0.000} C_DIS
LIN {X -26.261,Y 28.575,Z -184.848,A 90.000,B 90.000,C 0.000} C_DIS
LIN {X -24.831,Y 28.575,Z -183.529,A 90.000,B 90.000,C 0.000} C_DIS
LIN {X -23.438,Y 28.575,Z -182.171,A 90.000,B 90.000,C 0.000} C_DIS
LIN {X -144.015,Y 28.575,Z -182.171,A 90.000,B 90.000,C 0.000} C_DIS
LIN {X -144.015,Y 28.575,Z -174.622,A 90.000,B 90.000,C 0.000} C_DIS
LIN {X -16.895,Y 28.575,Z -174.622,A 90.000,B 90.000,C 0.000} C_DIS
LIN {X -15.936,Y 28.575,Z -173.314,A 90.000,B 90.000,C 0.000} C_DIS
LIN {X -15.007,Y 28.575,Z -171.984,A 90.000,B 90.000,C 0.000} C_DIS
LIN {X -14.422,Y 28.575,Z -171.056,A 90.000,B 90.000,C 0.000} C_DIS
LIN {X -13.887,Y 28.575,Z -170.098,A 90.000,B 90.000,C 0.000} C_DIS
LIN {X -13.405,Y 28.575,Z -169.113,A 90.000,B 90.000,C 0.000} C_DIS
LIN {X -12.975,Y 28.575,Z -168.104,A 90.000,B 90.000,C 0.000} C_DIS
LIN {X -12.600,Y 28.575,Z -167.073,A 90.000,B 90.000,C 0.000} C_DIS
LIN {X -144.015,Y 28.575,Z -167.073,A 90.000,B 90.000,C 0.000} C_DIS
LIN {X -144.015,Y 28.575,Z -159.525,A 90.000,B 90.000,C 0.000} C_DIS
LIN {X -18.930,Y 28.575,Z -159.525,A 90.000,B 90.000,C 0.000} C_DIS
LIN {X -20.483,Y 28.575,Z -158.329,A 90.000,B 90.000,C 0.000} C_DIS
LIN {X -22.044,Y 28.575,Z -157.142,A 90.000,B 90.000,C 0.000} C_DIS
LIN {X -24.030,Y 28.575,Z -155.458,A 90.000,B 90.000,C 0.000} C_DIS
LIN {X -25.983,Y 28.575,Z -153.735,A 90.000,B 90.000,C 0.000} C_DIS
LIN {X -27.902,Y 28.575,Z -151.976,A 90.000,B 90.000,C 0.000} C_DIS
LIN {X -144.015,Y 28.575,Z -151.976,A 90.000,B 90.000,C 0.000} C_DIS
LIN {X -144.015,Y 28.575,Z -144.427,A 90.000,B 90.000,C 0.000} C_DIS
LIN {X -35.097,Y 28.575,Z -144.427,A 90.000,B 90.000,C 0.000} C_DIS
LIN {X -35.914,Y 28.575,Z -143.370,A 90.000,B 90.000,C 0.000} C_DIS
LIN {X -36.708,Y 28.575,Z -142.295,A 90.000,B 90.000,C 0.000} C_DIS
LIN {X -37.476,Y 28.575,Z -141.202,A 90.000,B 90.000,C 0.000} C_DIS
LIN {X -38.365,Y 28.575,Z -140.156,A 90.000,B 90.000,C 0.000} C_DIS
LIN {X -39.225,Y 28.575,Z -139.087,A 90.000,B 90.000,C 0.000} C_DIS
LIN {X -40.055,Y 28.575,Z -137.994,A 90.000,B 90.000,C 0.000} C_DIS
LIN {X -40.854,Y 28.575,Z -136.878,A 90.000,B 90.000,C 0.000} C_DIS
LIN {X -144.015,Y 28.575,Z -136.878,A 90.000,B 90.000,C 0.000} C_DIS
LIN {X -144.015,Y 28.575,Z -129.329,A 90.000,B 90.000,C 0.000} C_DIS
